// Mitsubishi GX Works2 project: GHEP-Q02U-NEW   PLC: Q02U

// global labels: Global1
VAR_GLOBAL
  Servo_Ready_T AT X40 : BOOL;
  Servo_Ready_X1 AT X41 : BOOL;
  Servo_Ready_X2 AT X42 : BOOL;
  Servo_Ready_Ms AT X43 : BOOL;
  Servo_Ready_S AT X44 : BOOL;
  Physical_Start_PB AT X45 : BOOL;
  Physical_Stop_PB AT X46 : BOOL;
  Physical_Inc_PB AT X47 : BOOL;
  Physical_Dec_PB AT X48 : BOOL;
  Physical_Jog_PB AT X49 : BOOL;
  Sensor_Rev_M AT X4A : BOOL;
  Sensor_Rev_U AT X4B : BOOL;
  Pen1_Toggle_PB AT X4C : BOOL;
  Pen2_Toggle_PB AT X4D : BOOL;
  Switch_Hold_M AT X4E : BOOL;
  Switch_Hold_U AT X4F : BOOL;
  Servo_ON_T AT Y50 : BOOL;
  Servo_ON_X1 AT Y51 : BOOL;
  Servo_ON_X2 AT Y52 : BOOL;
  Servo_ON_Ms AT Y53 : BOOL;
  Servo_ON_S AT Y54 : BOOL;
  DO_Pen1 AT Y55 : BOOL;
  DO_Pen2 AT Y56 : BOOL;
  DO_Alarm_Horn AT Y57 : BOOL;
  Tower_Light_Green AT Y58 : BOOL;
  Tower_Light_Yellow AT Y59 : BOOL;
  Tower_Light_Red AT Y5A : BOOL;
  HMI_Auto_Mode AT M0 : BOOL;
  HMI_Reset_Error AT M1 : BOOL;
  HMI_Start AT M2 : BOOL;
  HMI_Stop AT M3 : BOOL;
  HMI_Reset_Length AT M4 : BOOL;
  HMI_Reset_Roll_T AT M5 : BOOL;
  HMI_Reset_Roll_M AT M6 : BOOL;
  HMI_Reset_Roll_U AT M7 : BOOL;
  HMI_Reset_All_Rolls AT M8 : BOOL;
  HMI_PID_Enable AT M9 : BOOL;
  HMI_Inc_Hold AT M10 : BOOL;
  HMI_Dec_Hold AT M11 : BOOL;
  HMI_Pen1_Cmd AT M12 : BOOL;
  HMI_Pen2_Cmd AT M13 : BOOL;
  HMI_Jog_Crawl_Cmd AT M14 : BOOL;
  HMI_Cmd_Apply_Recipe AT M15 : BOOL;
  HMI_Cmd_Save_Recipe AT M16 : BOOL;
  Zero_Set_T AT M20 : BOOL;
  Zero_Set_X1 AT M21 : BOOL;
  Zero_Set_M AT M22 : BOOL;
  Zero_Set_U AT M23 : BOOL;
  Calib_Set_T AT M24 : BOOL;
  Calib_Set_X1 AT M25 : BOOL;
  Calib_Set_M AT M26 : BOOL;
  Calib_Set_U AT M27 : BOOL;
  HMI_Cmd_Zero_Set AT M28 : BOOL;
  HMI_Cmd_Calib_Set AT M29 : BOOL;
  HMI_Test_T AT M30 : BOOL;
  HMI_Test_X1 AT M31 : BOOL;
  HMI_Test_X2 AT M32 : BOOL;
  HMI_Test_Ms AT M33 : BOOL;
  HMI_Test_S AT M34 : BOOL;
  HMI_Test_M AT M35 : BOOL;
  HMI_Test_U AT M36 : BOOL;
  HMI_Cmd_AutoTune AT M40 : BOOL;
  HMI_Cmd_Save_PID AT M41 : BOOL;
  HMI_Status_AT_Busy AT M42 : BOOL;
  HMI_Status_AT_Done AT M43 : BOOL;
  Servo_Not_Ready_Fault AT M50 : BOOL;
  Hold_Torque_Stop_M AT M51 : BOOL;
  Hold_Torque_Stop_U AT M52 : BOOL;
  Pen1_State AT M53 : BOOL;
  Pen2_State AT M54 : BOOL;
  Pen_Auto_Engaged AT M55 : BOOL;
  Auto_Decel_Flag AT M56 : BOOL;
  State_Machine AT D0 : INT;
  HMI_Status_Text_Code AT D1 : INT;
  HMI_Recipe_Select AT D2 : INT;
  Prev_Recipe_Select AT D3 : INT;
  Current_Line_MPM AT D10 : REAL;
  Total_Length_Meters AT D12 : REAL;
  Set_Target_Length AT D14 : REAL;
  Effective_SP_T AT D16 : REAL;
  RPM_T AT D50 : REAL;
  RPM_X1 AT D52 : REAL;
  RPM_X2 AT D54 : REAL;
  RPM_Ms AT D56 : REAL;
  RPM_S AT D58 : REAL;
  MPM_T AT D60 : REAL;
  MPM_X1 AT D62 : REAL;
  MPM_X2 AT D64 : REAL;
  MPM_Ms AT D66 : REAL;
  MPM_S AT D68 : REAL;
  Target_Line_MPM AT D100 : REAL;
  Max_Speed_MPM AT D102 : REAL;
  Min_Speed_MPM AT D104 : REAL;
  Release_Pen_Speed_MPM AT D106 : REAL;
  Ramp_Accel_Rate AT D108 : REAL;
  Ramp_Decel_Rate AT D110 : REAL;
  Decel_Distance_Meters AT D112 : REAL;
  SP_Tension_T AT D120 : REAL;
  SP_Tension_X1 AT D122 : REAL;
  SP_Tension_M AT D124 : REAL;
  SP_Tension_U AT D126 : REAL;
  Taper_Percent_T AT D128 : REAL;
  Gear_Ratio_T AT D200 : REAL;
  Gear_Ratio_X1 AT D202 : REAL;
  Gear_Ratio_X2 AT D204 : REAL;
  Gear_Ratio_Ms AT D206 : REAL;
  Gear_Ratio_S AT D208 : REAL;
  Gear_Ratio_U AT D210 : REAL;
  Max_RPM_T AT D212 : REAL;
  Max_RPM_X1 AT D214 : REAL;
  Max_RPM_X2 AT D216 : REAL;
  Max_RPM_Ms AT D218 : REAL;
  Max_RPM_S AT D220 : REAL;
  Dia_X1_Roller_mm AT D222 : REAL;
  Dia_X2_Roller_mm AT D224 : REAL;
  Dia_Ms_Roller_mm AT D226 : REAL;
  Dia_S_Roller_mm AT D228 : REAL;
  Core_Dia_T_mm AT D230 : REAL;
  Core_Dia_M_mm AT D232 : REAL;
  Core_Dia_U_mm AT D234 : REAL;
  Max_Dia_T_mm AT D236 : REAL;
  Max_Dia_M_mm AT D238 : REAL;
  Max_Dia_U_mm AT D240 : REAL;
  Speed_Ratio_T AT D250 : REAL;
  Speed_Ratio_X1 AT D252 : REAL;
  Speed_Ratio_Ms AT D254 : REAL;
  Speed_Ratio_S AT D256 : REAL;
  Speed_Offset_X1 AT D260 : REAL;
  Speed_Offset_Ms AT D262 : REAL;
  Speed_Offset_S AT D264 : REAL;
  Min_Torque_M AT D270 : REAL;
  Max_Torque_M AT D272 : REAL;
  Init_Holding_Torque_M AT D274 : REAL;
  Min_Torque_U AT D276 : REAL;
  Max_Torque_U AT D278 : REAL;
  Init_Holding_Torque_U AT D280 : REAL;
  Gear_Ratio_M AT D282 : REAL;
  PPR_Encoder AT D290 : DINT;
  Zero_Offset_T AT D300 : REAL;
  Zero_Offset_X1 AT D302 : REAL;
  Zero_Offset_M AT D304 : REAL;
  Zero_Offset_U AT D306 : REAL;
  Calib_Gain_T AT D310 : REAL;
  Calib_Gain_X1 AT D312 : REAL;
  Calib_Gain_M AT D314 : REAL;
  Calib_Gain_U AT D316 : REAL;
  Weight_Net_T AT D320 : REAL;
  Weight_Net_X1 AT D322 : REAL;
  Weight_Net_M AT D324 : REAL;
  Weight_Net_U AT D326 : REAL;
  Real_Dia_T_mm AT D330 : REAL;
  Real_Dia_M_mm AT D332 : REAL;
  Real_Dia_U_mm AT D334 : REAL;
  Kp_T AT D340 : REAL;
  Ki_T AT D342 : REAL;
  Kd_T AT D344 : REAL;
  Kp_X1 AT D346 : REAL;
  Ki_X1 AT D348 : REAL;
  Kd_X1 AT D350 : REAL;
  Kp_X2 AT D352 : REAL;
  Ki_X2 AT D354 : REAL;
  Kd_X2 AT D356 : REAL;
  Kp_Ms AT D358 : REAL;
  Ki_Ms AT D360 : REAL;
  Kd_Ms AT D362 : REAL;
  Kp_S AT D364 : REAL;
  Ki_S AT D366 : REAL;
  Kd_S AT D368 : REAL;
  Kp_M AT D370 : REAL;
  Ki_M AT D372 : REAL;
  Kd_M AT D374 : REAL;
  Kp_U AT D376 : REAL;
  Ki_U AT D378 : REAL;
  Kd_U AT D380 : REAL;
  Curr_Pulse_T AT D520 : DINT;
  Curr_Pulse_X1 AT D522 : DINT;
  Curr_Pulse_X2 AT D524 : DINT;
  Curr_Pulse_Ms AT D526 : DINT;
  HMI_Axis_Select AT D600 : INT;
  HMI_Disp_Kp AT D602 : REAL;
  HMI_Disp_Ki AT D604 : REAL;
  HMI_Disp_Kd AT D606 : REAL;
  HMI_Disp_Calib_Gain AT D608 : REAL;
  HMI_Disp_Zero_Offset AT D610 : REAL;
  Test_Speed_T AT D620 : REAL;
  Test_Torque_T AT D622 : REAL;
  Test_Speed_X1 AT D624 : REAL;
  Test_Speed_X2 AT D626 : REAL;
  Test_Speed_Ms AT D628 : REAL;
  Test_Speed_S AT D630 : REAL;
  Test_Torque_M AT D632 : REAL;
  Test_Speed_U AT D634 : REAL;
END_VAR

// task Task_01 (event TRUE, interval 0, priority 31): POU_01
// task POU_INIT (event TRUE, interval 0, priority 31): POU_INIT

PROGRAM POU_01
VAR
  Delta_T : DINT;  (* Chenh lech xung Truc Thu T *)
  Delta_X1 : DINT;  (* Chenh lech xung Truc Keo X1 *)
  Delta_X2 : DINT;  (* Chenh lech xung Master X2 *)
  Delta_Ms : DINT;  (* Chenh lech xung Truc Ghep Ms *)
  Delta_Pulse_X2 : DINT;  (* Chenh lech xung Master X2 tinh chieu dai mang *)
  Prev_Pulse_T : DINT;  (* Xung Truc T chu ky truoc *)
  Prev_Pulse_X1 : DINT;  (* Xung Truc X1 chu ky truoc *)
  Prev_Pulse_X2 : DINT;  (* Xung Truc X2 chu ky truoc *)
  Prev_Pulse_Ms : DINT;  (* Xung Truc Ms chu ky truoc *)
  Total_PPR : DINT;  (* Tong xung sau khi nhan 4 *)
  Raw_Analog_S : REAL;  (* Gia tri tho Analog Speed Servo S *)
  Raw_RPM_T : REAL;  (* Toc do RPM tho Truc Thu T *)
  Raw_RPM_X1 : REAL;  (* Toc do RPM tho Truc Keo X1 *)
  Raw_RPM_X2 : REAL;  (* Toc do RPM tho Truc Master X2 *)
  Raw_RPM_Ms : REAL;  (* Toc do RPM tho Truc Ghep Ms *)
  Raw_RPM_S : REAL;  (* Toc do RPM tho Truc Dau S *)
  Buf_RPM_T_1 : REAL;  (* Buffer mau 1 loc trung binh trượt T *)
  Buf_RPM_T_2 : REAL;  (* Buffer mau 2 loc trung binh trượt T *)
  Buf_RPM_T_3 : REAL;  (* Buffer mau 3 loc trung binh trượt T *)
  Buf_RPM_X1_1 : REAL;  (* Buffer mau 1 loc trung binh trượt X1 *)
  Buf_RPM_X1_2 : REAL;  (* Buffer mau 2 loc trung binh trượt X1 *)
  Buf_RPM_X1_3 : REAL;  (* Buffer mau 3 loc trung binh trượt X1 *)
  Buf_RPM_X2_1 : REAL;  (* Buffer mau 1 loc trung binh trượt X2 *)
  Buf_RPM_X2_2 : REAL;  (* Buffer mau 2 loc trung binh trượt X2 *)
  Buf_RPM_X2_3 : REAL;  (* Buffer mau 3 loc trung binh trượt X2 *)
  Buf_RPM_Ms_1 : REAL;  (* Buffer mau 1 loc trung binh trượt Ms *)
  Buf_RPM_Ms_2 : REAL;  (* Buffer mau 2 loc trung binh trượt Ms *)
  Buf_RPM_Ms_3 : REAL;  (* Buffer mau 3 loc trung binh trượt Ms *)
  Buf_RPM_S_1 : REAL;  (* Buffer mau 1 loc trung binh trượt S *)
  Buf_RPM_S_2 : REAL;  (* Buffer mau 2 loc trung binh trượt S *)
  Buf_RPM_S_3 : REAL;  (* Buffer mau 3 loc trung binh trượt S *)
  ADC_CH1_Raw : INT;  (* Gia tri tho ADC CH1 Loadcell T *)
  ADC_CH2_Raw : INT;  (* Gia tri tho ADC CH2 Loadcell X1 *)
  ADC_CH3_Raw : INT;  (* Gia tri tho ADC CH3 Loadcell M *)
  ADC_CH4_Raw : INT;  (* Gia tri tho ADC CH4 Loadcell U *)
  ADC_CH5_Raw : INT;  (* Gia tri tho ADC CH5 Analog Servo S *)
  ADC_CH6_Raw : INT;  (* Gia tri tho ADC CH6 Du phong *)
  ADC_CH7_Raw : INT;  (* Gia tri tho ADC CH7 Du phong *)
  ADC_CH8_Raw : INT;  (* Gia tri tho ADC CH8 Du phong *)
  Cmd_Start : BOOL;  (* Lenh tong hop Start chay may *)
  Cmd_Stop : BOOL;  (* Lenh tong hop Stop dung may *)
  Cmd_Inc : BOOL;  (* Lenh tong hop Tang toc *)
  Cmd_Dec : BOOL;  (* Lenh tong hop Giam toc *)
  Cmd_Jog_Crawl : BOOL;  (* Lenh tong hop Bo cham luon mang *)
  Trig_Pen1 : BOOL;  (* Xung kich toggle Pen 1 *)
  Prev_Pen1_PB : BOOL;  (* Trang thai Pen 1 chu ky truoc *)
  Trig_Pen2 : BOOL;  (* Xung kich toggle Pen 2 *)
  Prev_Pen2_PB : BOOL;  (* Trang thai Pen 2 chu ky truoc *)
  Pen1_Next_State : BOOL;  (* Trang thai tiep theo Pen 1 *)
  Pen2_Next_State : BOOL;  (* Trang thai tiep theo Pen 2 *)
  Trig_X50 : BOOL;  (* Xung kich sensor cuon M *)
  Prev_X50 : BOOL;  (* Trang thai sensor cuon M chu ky truoc *)
  Trig_X51 : BOOL;  (* Xung kich sensor cuon U *)
  Prev_X51 : BOOL;  (* Trang thai sensor cuon U chu ky truoc *)
  Trig_PID_10ms : BOOL;  (* Xung kich nhap PID 10ms *)
  Prev_SM409 : BOOL;  (* Trang thai SM409 chu ky truoc *)
  Inc_Hold_Timer : INT;  (* Timer giu nut tang toc *)
  Dec_Hold_Timer : INT;  (* Timer giu nut giam toc *)
  Dynamic_Accel_Step : REAL;  (* Buoc tang giam toc luy tien *)
  Last_Pulse_X2_Len : DINT;  (* Xung X2 chu ky truoc tinh chieu dai *)
  Last_Pulse_X2_T : DINT;  (* Xung X2 chu ky truoc tinh duong kinh T *)
  Last_Pulse_X2_M : DINT;  (* Xung X2 chu ky truoc tinh duong kinh M *)
  Last_Pulse_X2_U : DINT;  (* Xung X2 chu ky truoc tinh duong kinh U *)
  Last_Pulse_T : DINT;  (* Xung T chu ky truoc *)
  Rev_Count_T : DINT;  (* So vong quay cuon Thu T *)
  Rev_Count_M : DINT;  (* So vong quay cuon Thang M *)
  Rev_Count_U : DINT;  (* So vong quay cuon Xa U *)
  Accum_Length_mm : REAL;  (* Chieu dai tich luy mm *)
  Delta_Length_mm : REAL;  (* Chieu dai di duoc trong 1 scan mm *)
  Raw_Dia_T_mm : REAL;  (* Duong kinh tho tinh toan T mm *)
  Raw_Dia_M_mm : REAL;  (* Duong kinh tho tinh toan M mm *)
  Raw_Dia_U_mm : REAL;  (* Duong kinh tho tinh toan U mm *)
  Base_Speed_X2 : REAL;  (* Toc do co ban theo Master X2 (0..16000) *)
  SP_Speed_X2 : REAL;  (* Setpoint toc do Master X2 *)
  SP_Speed_X1 : REAL;  (* Setpoint toc do Keo X1 *)
  SP_Speed_Ms : REAL;  (* Setpoint toc do Ghep Ms *)
  SP_Speed_S : REAL;  (* Setpoint toc do Dau S *)
  SP_Speed_T : REAL;  (* Setpoint toc do Thu T *)
  Feedback_Speed_X2 : REAL;  (* Feedback toc do Master X2 *)
  Feedback_Speed_Ms : REAL;  (* Feedback toc do Ghep Ms *)
  Feedback_Speed_S : REAL;  (* Feedback toc do Dau S (tu Analog Out Servo) *)
  PID_Out_X2 : REAL;  (* Ngo ra PID Master X2 *)
  PID_Out_Ms : REAL;  (* Ngo ra PID Ghep Ms *)
  PID_Out_S : REAL;  (* Ngo ra PID Dau S *)
  PID_Out_X1 : REAL;  (* Ngo ra PID Keo X1 *)
  PID_Out_T : REAL;  (* Ngo ra PID Thu T *)
  PID_Out_M : REAL;  (* Ngo ra PID Thang M *)
  PID_Out_U : REAL;  (* Ngo ra PID Xa U *)
  Calc_Speed_X2 : REAL;  (* Toc do tong hop xuat DAC Master X2 *)
  Calc_Speed_X1 : REAL;  (* Toc do tong hop xuat DAC Keo X1 *)
  Calc_Speed_Ms : REAL;  (* Toc do tong hop xuat DAC Ghep Ms *)
  Calc_Speed_S : REAL;  (* Toc do tong hop xuat DAC Dau S *)
  Calc_Speed_T : REAL;  (* Toc do tong hop xuat DAC Thu T *)
  Calc_Speed_U : REAL;  (* Toc do tong hop xuat DAC Xa U *)
  Calc_Torque_T : REAL;  (* Torque tong hop xuat DAC Thu T *)
  Calc_Torque_M : REAL;  (* Torque tong hop xuat DAC Thang M *)
  Base_Torque_M : REAL;  (* Torque co ban 3 pha Thang M (%) *)
  pid_X2 : FB_TENSION_PID;  (* Instance PID Master X2 *)
  pid_Ms : FB_TENSION_PID;  (* Instance PID Ghep Ms *)
  pid_S : FB_TENSION_PID;  (* Instance PID Dau S *)
  pid_X1 : FB_TENSION_PID;  (* Instance PID Keo X1 *)
  pid_T : FB_TENSION_PID;  (* Instance PID Thu T *)
  pid_M : FB_TENSION_PID;  (* Instance PID Thang M *)
  pid_U : FB_TENSION_PID;  (* Instance PID Xa U *)
END_VAR
(* ============================================================================ *)
(* MÃ NGUỒN POU_01: HỆ THỐNG MÁY GHÉP MÀNG METALIZE TỰ ĐỘNG - MITSUBISHI Q02U  *)
(* BẢO VỆ TOÀN DIỆN CHỐNG LỖI 4140 OPERATION ERROR (CHIA CHO 0 & TRÀN SỐ DINT)  *)
(* CẤU HÌNH PHẦN CỨNG:                                                          *)
(*   - Slot 0 (H00): Q68ADV (8CH Analog In: Loadcell T, X1, M, U & Analog S)    *)
(*   - Slot 1 (H10): Q68DAV (8CH Analog Out: Speed/Torque T, X1, X2, Ms, S, M, U) *)
(*   - Slot 2 (H20): QD62D  (2CH High Speed Counter: CH1=Trục T, CH2=Trục X1)  *)
(*   - Slot 3 (H30): QD62D  (2CH High Speed Counter: CH1=Trục X2, CH2=Trục Ms) *)
(*   - Slot 4 (H40): QX40   (16CH Digital Input: X40..X4F)                     *)
(*   - Slot 5 (H50): QY40   (16CH Digital Output: Y50..Y5F)                    *)
(*   - Slot 6 (H60): QJ71C24N (RS232/RS485 Serial)                             *)
(* ============================================================================ *)

(* ============================================================================ *)
(* 0. KIỂM TRA & GÁN GIÁ TRỊ AN TOÀN TRÁNH CHIA CHO 0 (ZERO DIV PROTECTION)    *)
(* ============================================================================ *)
IF PPR_Encoder      <= 0     THEN PPR_Encoder      := 2000;  END_IF;
IF Max_RPM_X2       <= 0.0   THEN Max_RPM_X2       := 1000.0; END_IF;
IF Max_RPM_X1       <= 0.0   THEN Max_RPM_X1       := 1000.0; END_IF;
IF Max_RPM_Ms       <= 0.0   THEN Max_RPM_Ms       := 3000.0; END_IF;
IF Max_RPM_S        <= 0.0   THEN Max_RPM_S        := 3000.0; END_IF;
IF Max_RPM_T        <= 0.0   THEN Max_RPM_T        := 1500.0; END_IF;

IF Gear_Ratio_T     <= 0.0   THEN Gear_Ratio_T     := 10.1;  END_IF;
IF Gear_Ratio_X1    <= 0.0   THEN Gear_Ratio_X1    := 8.0;   END_IF;
IF Gear_Ratio_X2    <= 0.0   THEN Gear_Ratio_X2    := 8.0;   END_IF;
IF Gear_Ratio_Ms    <= 0.0   THEN Gear_Ratio_Ms    := 10.0;  END_IF;
IF Gear_Ratio_S     <= 0.0   THEN Gear_Ratio_S     := 10.0;  END_IF;
IF Gear_Ratio_U     <= 0.0   THEN Gear_Ratio_U     := 1.0;     END_IF; (* Xả U: 1.0 : 1 *)
IF Gear_Ratio_M     <= 0.0   THEN Gear_Ratio_M     := 1.03125; END_IF; (* Trục Xả Metalize M: Gear = 33/32 = 1.03125 *)

IF Dia_X1_Roller_mm <= 0.0   THEN Dia_X1_Roller_mm := 300.5; END_IF;
IF Dia_X2_Roller_mm <= 0.0   THEN Dia_X2_Roller_mm := 300.5; END_IF;
IF Dia_Ms_Roller_mm <= 0.0   THEN Dia_Ms_Roller_mm := 200.0; END_IF;
IF Dia_S_Roller_mm  <= 0.0   THEN Dia_S_Roller_mm  := 100.0; END_IF;

IF Core_Dia_T_mm    <= 0.0   THEN Core_Dia_T_mm    := 76.0;   END_IF;
IF Core_Dia_M_mm    <= 0.0   THEN Core_Dia_M_mm    := 76.0;   END_IF;
IF Core_Dia_U_mm    <= 0.0   THEN Core_Dia_U_mm    := 76.0;   END_IF;

IF Max_Dia_T_mm     <= 0.0   THEN Max_Dia_T_mm     := 1000.0; END_IF;
IF Max_Dia_M_mm     <= 0.0   THEN Max_Dia_M_mm     := 600.0;  END_IF;
IF Max_Dia_U_mm     <= 0.0   THEN Max_Dia_U_mm     := 800.0;  END_IF;

IF Real_Dia_T_mm    < Core_Dia_T_mm THEN Real_Dia_T_mm := Core_Dia_T_mm; END_IF;
IF Real_Dia_M_mm    < Core_Dia_M_mm THEN Real_Dia_M_mm := Max_Dia_M_mm;  END_IF;
IF Real_Dia_U_mm    < Core_Dia_U_mm THEN Real_Dia_U_mm := Max_Dia_U_mm;  END_IF;

IF Max_Speed_MPM    <= 0.0   THEN Max_Speed_MPM    := 100.0;  END_IF;
IF Min_Speed_MPM    <= 0.0   THEN Min_Speed_MPM    := 2.0;    END_IF;
IF Ramp_Accel_Rate  <= 0.0   THEN Ramp_Accel_Rate  := 0.5;    END_IF;
IF Ramp_Decel_Rate  <= 0.0   THEN Ramp_Decel_Rate  := 1.0;    END_IF;

(* ============================================================================ *)
(* 1. KÍCH HOẠT VÀ ĐỌC 4 KÊNH ENCODER QD62D (SLOT 2 & 3) MỖI SCAN               *)
(* ============================================================================ *)
(* Kích hoạt cờ đếm xung cho 2 module QD62D *)
Y21 := TRUE; (* QD62D #1 (Slot 2 H20) CH1: Enable Trục Thu T *)
Y22 := TRUE; (* QD62D #1 (Slot 2 H20) CH2: Enable Trục Kéo X1 *)
Y31 := TRUE; (* QD62D #2 (Slot 3 H30) CH1: Enable Trục Master X2 *)
Y32 := TRUE; (* QD62D #2 (Slot 3 H30) CH2: Enable Trục Ghép Ms *)

(* Đọc xung 32-bit từ Buffer Memory QD62D liên tục mỗi scan *)
DMOV(TRUE, U2\G2,  Curr_Pulse_T);  (* Slot 2 CH1: Trục Thu T *)
DMOV(TRUE, U2\G10, Curr_Pulse_X1); (* Slot 2 CH2: Trục Kéo X1 *)
DMOV(TRUE, U3\G2,  Curr_Pulse_X2); (* Slot 3 CH1: Trục Master X2 *)
DMOV(TRUE, U3\G10, Curr_Pulse_Ms); (* Slot 3 CH2: Trục Ghép Ms *)

(* ============================================================================ *)
(* 2. ĐỌC VÀ LỌC 8 KÊNH ANALOG INPUT TỪ MODULE Q68ADV (SLOT 0 - U0\G1..U0\G8)   *)
(* ============================================================================ *)
ADC_CH1_Raw := U0\G1; (* Loadcell Lực căng Thu T *)
ADC_CH2_Raw := U0\G2; (* Loadcell Lực căng Kéo X1 *)
ADC_CH3_Raw := U0\G3; (* Loadcell Lực căng Thắng M *)
ADC_CH4_Raw := U0\G4; (* Loadcell Lực căng Xả U *)
ADC_CH5_Raw := U0\G5; (* Tín hiệu Analog Out Tốc độ Servo Trục S *)
ADC_CH6_Raw := U0\G6; (* Dự phòng CH6 *)
ADC_CH7_Raw := U0\G7; (* Dự phòng CH7 *)
ADC_CH8_Raw := U0\G8; (* Dự phòng CH8 *)

(* Chuyển sang thanh ghi hiển thị D500..D507 *)
D500 := INT_TO_WORD(ADC_CH1_Raw);
D501 := INT_TO_WORD(ADC_CH2_Raw);
D502 := INT_TO_WORD(ADC_CH3_Raw);
D503 := INT_TO_WORD(ADC_CH4_Raw);
D504 := INT_TO_WORD(ADC_CH5_Raw);
D505 := INT_TO_WORD(ADC_CH6_Raw);
D506 := INT_TO_WORD(ADC_CH7_Raw);
D507 := INT_TO_WORD(ADC_CH8_Raw);

(* Tính giá trị Lực căng thực tế (kg) sau khi trừ Zero Offset và nhân Gain Calib *)
IF Calib_Gain_T <= 0.0 THEN Calib_Gain_T := 1.0; END_IF;
Weight_Net_T := ((INT_TO_REAL(ADC_CH1_Raw) - Zero_Offset_T) * Calib_Gain_T * 50.0) / 16000.0;
IF Weight_Net_T < 0.0 THEN Weight_Net_T := 0.0; END_IF;

IF Calib_Gain_X1 <= 0.0 THEN Calib_Gain_X1 := 1.0; END_IF;
Weight_Net_X1 := ((INT_TO_REAL(ADC_CH2_Raw) - Zero_Offset_X1) * Calib_Gain_X1 * 50.0) / 16000.0;
IF Weight_Net_X1 < 0.0 THEN Weight_Net_X1 := 0.0; END_IF;

IF Calib_Gain_M <= 0.0 THEN Calib_Gain_M := 1.0; END_IF;
Weight_Net_M := ((INT_TO_REAL(ADC_CH3_Raw) - Zero_Offset_M) * Calib_Gain_M * 50.0) / 16000.0;
IF Weight_Net_M < 0.0 THEN Weight_Net_M := 0.0; END_IF;

IF Calib_Gain_U <= 0.0 THEN Calib_Gain_U := 1.0; END_IF;
Weight_Net_U := ((INT_TO_REAL(ADC_CH4_Raw) - Zero_Offset_U) * Calib_Gain_U * 50.0) / 16000.0;
IF Weight_Net_U < 0.0 THEN Weight_Net_U := 0.0; END_IF;

(* Xử lý Nút Set Zero Lực căng *)
IF Zero_Set_T OR (HMI_Cmd_Zero_Set AND HMI_Axis_Select = 1) THEN
    Zero_Offset_T := INT_TO_REAL(ADC_CH1_Raw);
    Zero_Set_T    := FALSE;
END_IF;
IF Zero_Set_X1 OR (HMI_Cmd_Zero_Set AND HMI_Axis_Select = 2) THEN
    Zero_Offset_X1 := INT_TO_REAL(ADC_CH2_Raw);
    Zero_Set_X1    := FALSE;
END_IF;
IF Zero_Set_M OR (HMI_Cmd_Zero_Set AND HMI_Axis_Select = 6) THEN
    Zero_Offset_M := INT_TO_REAL(ADC_CH3_Raw);
    Zero_Set_M    := FALSE;
END_IF;
IF Zero_Set_U OR (HMI_Cmd_Zero_Set AND HMI_Axis_Select = 7) THEN
    Zero_Offset_U := INT_TO_REAL(ADC_CH4_Raw);
    Zero_Set_U    := FALSE;
END_IF;
IF HMI_Cmd_Zero_Set THEN
    HMI_Cmd_Zero_Set := FALSE;
END_IF;

(* ============================================================================ *)
(* 3. BẢO VỆ 5 TRỤC SERVO READY TRÊN MODULE QX40 (SLOT 4 - X40..X44)            *)
(* ============================================================================ *)
Servo_Ready_T  := X40; (* Sẵn sàng Servo Thu T *)
Servo_Ready_X1 := X41; (* Sẵn sàng Servo Kéo X1 *)
Servo_Ready_X2 := X42; (* Sẵn sàng Servo Master X2 *)
Servo_Ready_Ms := X43; (* Sẵn sàng Servo Ghép Ms *)
Servo_Ready_S  := X44; (* Sẵn sàng Servo Dầu S *)

Servo_Not_Ready_Fault := NOT(Servo_Ready_T) OR NOT(Servo_Ready_X1) OR NOT(Servo_Ready_X2) OR NOT(Servo_Ready_Ms) OR NOT(Servo_Ready_S);

IF Servo_Not_Ready_Fault AND State_Machine = 1 THEN
    State_Machine := 0; (* Dừng khẩn cấp nếu đang chạy tự động *)
END_IF;

(* ============================================================================ *)
(* 4. ĐỌC NÚT NHẤN, CẢM BIẾN VÀ CÔNG TẮC GẠT TRÊN MODULE QX40 (SLOT 4 - X45..X4F) *)
(* ============================================================================ *)
Physical_Start_PB := X45; (* Nút Start vật lý *)
Physical_Stop_PB  := X46; (* Nút Stop vật lý *)
Physical_Inc_PB   := X47; (* Nút Tăng tốc vật lý *)
Physical_Dec_PB   := X48; (* Nút Giảm tốc vật lý *)
Physical_Jog_PB   := X49; (* Nút Bò chậm luồn màng vật lý *)
Sensor_Rev_M      := X4A; (* Cảm biến tiệm cận đếm vòng cuộn M *)
Sensor_Rev_U      := X4B; (* Cảm biến tiệm cận đếm vòng cuộn U *)
Pen1_Toggle_PB    := X4C; (* Nút nhấn Pen 1 ngoài tủ *)
Pen2_Toggle_PB    := X4D; (* Nút nhấn Pen 2 ngoài tủ *)
Switch_Hold_M     := X4E; (* Công tắc gạt giữ Torque M khi dừng *)
Switch_Hold_U     := X4F; (* Công tắc gạt giữ Torque U khi dừng *)

Hold_Torque_Stop_M := Switch_Hold_M;
Hold_Torque_Stop_U := Switch_Hold_U;

(* ============================================================================ *)
(* 5. QUẢN LÝ CÔNG THỨC ĐƠN HÀNG (RECIPE MANAGEMENT CHO CÔNG NHÂN)             *)
(* ============================================================================ *)
IF HMI_Recipe_Select <= 0 OR HMI_Recipe_Select > 5 THEN
    HMI_Recipe_Select := 2; (* Mặc định chọn Recipe 2: Hàng Tiêu Chuẩn *)
END_IF;

IF (HMI_Recipe_Select <> Prev_Recipe_Select) OR HMI_Cmd_Apply_Recipe THEN
    CASE HMI_Recipe_Select OF
        1: (* 1. HÀNG MÀNG MỎNG (BOPP 12~15 mic - Bao bì bánh kẹo) *)
            Target_Line_MPM  := 45.0;  (* Tốc độ chuẩn 45 m/p *)
            SP_Tension_T     := 12.0;  (* Lực căng Thu T: 12 kg *)
            SP_Tension_X1    := 10.0;  (* Lực căng Kéo X1: 10 kg *)
            SP_Tension_M     := 4.0;   (* Lực căng Thắng Metalize M: 4 kg *)
            SP_Tension_U     := 8.0;   (* Lực căng Xả U: 8 kg *)
            Taper_Percent_T  := 15.0;  (* Giảm côn lực 15% *)
            Ramp_Accel_Rate  := 0.05;  (* Gia tốc êm ái *)
            Ramp_Decel_Rate  := 0.08;

        2: (* 2. HÀNG TIÊU CHUẨN (BOPP 18~20 mic + Giấy 100~150g - Hộp thông dụng) *)
            Target_Line_MPM  := 60.0;  (* Tốc độ chuẩn 60 m/p *)
            SP_Tension_T     := 16.0;  (* Lực căng Thu T: 16 kg *)
            SP_Tension_X1    := 14.0;  (* Lực căng Kéo X1: 14 kg *)
            SP_Tension_M     := 6.0;   (* Lực căng Thắng Metalize M: 6 kg *)
            SP_Tension_U     := 12.0;  (* Lực căng Xả U: 12 kg *)
            Taper_Percent_T  := 20.0;  (* Giảm côn lực 20% *)
            Ramp_Accel_Rate  := 0.08;  (* Gia tốc tiêu chuẩn *)
            Ramp_Decel_Rate  := 0.10;

        3: (* 3. HÀNG GIẤY DÀY / BÌA CỨNG (Duplex / Ivory 250~350g + Metalize) *)
            Target_Line_MPM  := 50.0;  (* Tốc độ chuẩn 50 m/p *)
            SP_Tension_T     := 25.0;  (* Lực căng Thu T: 25 kg *)
            SP_Tension_X1    := 22.0;  (* Lực căng Kéo X1: 22 kg *)
            SP_Tension_M     := 8.0;   (* Lực căng Thắng Metalize M: 8 kg *)
            SP_Tension_U     := 18.0;  (* Lực căng Xả U: 18 kg *)
            Taper_Percent_T  := 25.0;  (* Giảm côn lực 25% *)
            Ramp_Accel_Rate  := 0.06;
            Ramp_Decel_Rate  := 0.10;

        4: (* 4. HÀNG MÀNG NHÔM / FOIL DẺO CAO CẤP (Alu Foil 9~12 mic / PET) *)
            Target_Line_MPM  := 40.0;  (* Tốc độ chuẩn 40 m/p *)
            SP_Tension_T     := 10.0;  (* Lực căng Thu T: 10 kg *)
            SP_Tension_X1    := 8.0;   (* Lực căng Kéo X1: 8 kg *)
            SP_Tension_M     := 3.5;   (* Lực căng Thắng Metalize M: 3.5 kg *)
            SP_Tension_U     := 7.0;   (* Lực căng Xả U: 7 kg *)
            Taper_Percent_T  := 15.0;
            Ramp_Accel_Rate  := 0.04;  (* Gia tốc siêu êm chống đứt foil *)
            Ramp_Decel_Rate  := 0.06;

        5: (* 5. CHẾ ĐỘ TÙY CHỈNH (CUSTOM) *)
            Target_Line_MPM := Target_Line_MPM;
    END_CASE;
    Prev_Recipe_Select   := HMI_Recipe_Select;
    HMI_Cmd_Apply_Recipe := FALSE;
END_IF;

IF HMI_Cmd_Save_Recipe THEN
    HMI_Recipe_Select    := 5;
    Prev_Recipe_Select   := 5;
    HMI_Cmd_Save_Recipe  := FALSE;
END_IF;

(* ============================================================================ *)
(* 6. NẠP LẠI ĐƯỜNG KÍNH CUỘN TỪ HMI & NÚT THAY CUỘN MỚI TOÀN BỘ 1-CLICK        *)
(* ============================================================================ *)
IF HMI_Reset_All_Rolls THEN
    Real_Dia_T_mm       := Core_Dia_T_mm; (* Thu T về lõi *)
    Real_Dia_M_mm       := Max_Dia_M_mm;  (* Thắng M về cuộn đầy *)
    Real_Dia_U_mm       := Max_Dia_U_mm;  (* Xả U về cuộn đầy *)
    Total_Length_Meters := 0.0;           (* Xóa mét về 0 *)
    Accum_Length_mm     := 0.0;
    HMI_Reset_All_Rolls := FALSE;
END_IF;
IF HMI_Reset_Roll_T THEN Real_Dia_T_mm := Core_Dia_T_mm; HMI_Reset_Roll_T := FALSE; END_IF;
IF HMI_Reset_Roll_M THEN Real_Dia_M_mm := Max_Dia_M_mm;  HMI_Reset_Roll_M := FALSE; END_IF;
IF HMI_Reset_Roll_U THEN Real_Dia_U_mm := Max_Dia_U_mm;  HMI_Reset_Roll_U := FALSE; END_IF;

(* ============================================================================ *)
(* 7. TỔNG HỢP NÚT NHẤN HMI & NÚT NHẤN VẬT LÝ                                  *)
(* ============================================================================ *)
Cmd_Start     := HMI_Start OR Physical_Start_PB;
Cmd_Stop      := HMI_Stop OR Physical_Stop_PB OR Servo_Not_Ready_Fault;
Cmd_Inc       := HMI_Inc_Hold OR Physical_Inc_PB;
Cmd_Dec       := HMI_Dec_Hold OR Physical_Dec_PB;
Cmd_Jog_Crawl := HMI_Jog_Crawl_Cmd OR Physical_Jog_PB;

(* ============================================================================ *)
(* 8. ĐIỀU KHIỂN 2 PEN ÉP MÀNG (SINGLE-COIL LOGIC)                             *)
(* ============================================================================ *)
Trig_Pen1 := (Pen1_Toggle_PB AND NOT(Prev_Pen1_PB)) OR HMI_Pen1_Cmd;
Prev_Pen1_PB := Pen1_Toggle_PB;
IF HMI_Pen1_Cmd THEN HMI_Pen1_Cmd := FALSE; END_IF;

Trig_Pen2 := (Pen2_Toggle_PB AND NOT(Prev_Pen2_PB)) OR HMI_Pen2_Cmd;
Prev_Pen2_PB := Pen2_Toggle_PB;
IF HMI_Pen2_Cmd THEN HMI_Pen2_Cmd := FALSE; END_IF;

IF State_Machine = 1 AND Current_Line_MPM >= 5.0 AND NOT Pen_Auto_Engaged THEN
    Pen1_Next_State := TRUE;
    Pen2_Next_State := TRUE;
ELSIF (State_Machine = 0 OR Current_Line_MPM <= Release_Pen_Speed_MPM) AND NOT (Trig_Pen1 OR Trig_Pen2) THEN
    Pen1_Next_State := FALSE;
    Pen2_Next_State := FALSE;
ELSE
    IF Trig_Pen1 THEN Pen1_Next_State := NOT Pen1_State; ELSE Pen1_Next_State := Pen1_State; END_IF;
    IF Trig_Pen2 THEN Pen2_Next_State := NOT Pen2_State; ELSE Pen2_Next_State := Pen2_State; END_IF;
END_IF;

Pen1_State := Pen1_Next_State;
Pen2_State := Pen2_Next_State;
Pen_Auto_Engaged := (State_Machine = 1 AND Current_Line_MPM >= 5.0);

(* ============================================================================ *)
(* 9. TĂNG GIẢM TỐC LŨY TIẾN THEO THỜI GIAN GIỮ PHÍM INC / DEC                 *)
(* ============================================================================ *)
IF Cmd_Inc THEN
    Inc_Hold_Timer := Inc_Hold_Timer + 1;
    IF Inc_Hold_Timer < 50 THEN
        Dynamic_Accel_Step := Ramp_Accel_Rate;
    ELSIF Inc_Hold_Timer < 150 THEN
        Dynamic_Accel_Step := Ramp_Accel_Rate * 2.0;
    ELSE
        Dynamic_Accel_Step := Ramp_Accel_Rate * 5.0;
    END_IF;
    Target_Line_MPM := Target_Line_MPM + Dynamic_Accel_Step;
    IF Target_Line_MPM > Max_Speed_MPM THEN Target_Line_MPM := Max_Speed_MPM; END_IF;
ELSE
    Inc_Hold_Timer := 0;
END_IF;

IF Cmd_Dec THEN
    Dec_Hold_Timer := Dec_Hold_Timer + 1;
    IF Dec_Hold_Timer < 50 THEN
        Dynamic_Accel_Step := Ramp_Decel_Rate;
    ELSIF Dec_Hold_Timer < 150 THEN
        Dynamic_Accel_Step := Ramp_Decel_Rate * 2.0;
    ELSE
        Dynamic_Accel_Step := Ramp_Decel_Rate * 5.0;
    END_IF;
    Target_Line_MPM := Target_Line_MPM - Dynamic_Accel_Step;
    IF Target_Line_MPM < Min_Speed_MPM THEN Target_Line_MPM := Min_Speed_MPM; END_IF;
ELSE
    Dec_Hold_Timer := 0;
END_IF;

(* Ramping tốc độ hiện tại *)
IF Current_Line_MPM < Target_Line_MPM THEN
    Current_Line_MPM := Current_Line_MPM + Ramp_Accel_Rate;
    IF Current_Line_MPM > Target_Line_MPM THEN Current_Line_MPM := Target_Line_MPM; END_IF;
ELSIF Current_Line_MPM > Target_Line_MPM THEN
    Current_Line_MPM := Current_Line_MPM - Ramp_Decel_Rate;
    IF Current_Line_MPM < Target_Line_MPM THEN Current_Line_MPM := Target_Line_MPM; END_IF;
END_IF;

(* ============================================================================ *)
(* 10. TÍNH ĐƯỜNG KÍNH 3 CUỘN T, M, U VÀ ĐO CHIỀU DÀI MÀNG CHẠY TỪ ENCODER X2   *)
(* ============================================================================ *)
Delta_Pulse_X2 := ABS(Curr_Pulse_X2 - Last_Pulse_X2_Len);

IF Delta_Pulse_X2 > 0 AND State_Machine = 1 AND Total_PPR > 0 THEN
    Delta_Length_mm := (DINT_TO_REAL(Delta_Pulse_X2) * 3.1415 * Dia_X2_Roller_mm) / (DINT_TO_REAL(Total_PPR) * Gear_Ratio_X2);
    Accum_Length_mm := Accum_Length_mm + Delta_Length_mm;
    
    IF Accum_Length_mm >= 1000.0 THEN
        Total_Length_Meters := Total_Length_Meters + (Accum_Length_mm / 1000.0);
        Accum_Length_mm     := 0.0;
    END_IF;
END_IF;
Last_Pulse_X2_Len := Curr_Pulse_X2;

IF HMI_Reset_Length THEN
    Total_Length_Meters := 0.0;
    Accum_Length_mm     := 0.0;
    HMI_Reset_Length    := FALSE;
END_IF;

(* Đường kính cuộn Thu T theo xung Master X2 *)
IF Total_PPR > 0 AND (Curr_Pulse_T - Last_Pulse_T) >= REAL_TO_DINT(DINT_TO_REAL(Total_PPR) * Gear_Ratio_T) THEN
    Rev_Count_T := Rev_Count_T + 1;
    IF (Curr_Pulse_X2 - Last_Pulse_X2_T) > 0 THEN
        Raw_Dia_T_mm := (DINT_TO_REAL(Curr_Pulse_X2 - Last_Pulse_X2_T) * Dia_X2_Roller_mm) / (DINT_TO_REAL(Total_PPR) * Gear_Ratio_X2);
        IF Raw_Dia_T_mm < Core_Dia_T_mm THEN Raw_Dia_T_mm := Core_Dia_T_mm; END_IF;
        IF Raw_Dia_T_mm > Max_Dia_T_mm THEN Raw_Dia_T_mm := Max_Dia_T_mm; END_IF;
        Real_Dia_T_mm := Real_Dia_T_mm + ((Raw_Dia_T_mm - Real_Dia_T_mm) * 0.2);
    END_IF;
    Last_Pulse_X2_T := Curr_Pulse_X2;
    Last_Pulse_T    := Curr_Pulse_T;
END_IF;

(* Đường kính cuộn Xả Metalize M theo cảm biến tiệm cận X4A & Tỷ số truyền Gear_Ratio_M (33/32) *)
Trig_X50 := Sensor_Rev_M AND NOT(Prev_X50);
Prev_X50 := Sensor_Rev_M;
IF Trig_X50 THEN
    Rev_Count_M := Rev_Count_M + 1;
    IF Total_PPR > 0 AND (Curr_Pulse_X2 - Last_Pulse_X2_M) > 0 THEN
        Raw_Dia_M_mm := (DINT_TO_REAL(Curr_Pulse_X2 - Last_Pulse_X2_M) * Dia_X2_Roller_mm * Gear_Ratio_M) / (DINT_TO_REAL(Total_PPR) * Gear_Ratio_X2);
        IF Raw_Dia_M_mm < Core_Dia_M_mm THEN Raw_Dia_M_mm := Core_Dia_M_mm; END_IF;
        IF Raw_Dia_M_mm > Max_Dia_M_mm THEN Raw_Dia_M_mm := Max_Dia_M_mm; END_IF;
        Real_Dia_M_mm := Real_Dia_M_mm + ((Raw_Dia_M_mm - Real_Dia_M_mm) * 0.2);
    END_IF;
    Last_Pulse_X2_M := Curr_Pulse_X2;
END_IF;

(* Đường kính cuộn Xả U theo cảm biến tiệm cận X4B *)
Trig_X51 := Sensor_Rev_U AND NOT(Prev_X51);
Prev_X51 := Sensor_Rev_U;
IF Trig_X51 THEN
    Rev_Count_U := Rev_Count_U + 1;
    IF Total_PPR > 0 AND (Curr_Pulse_X2 - Last_Pulse_X2_U) > 0 THEN
        Raw_Dia_U_mm := (DINT_TO_REAL(Curr_Pulse_X2 - Last_Pulse_X2_U) * Dia_X2_Roller_mm) / (DINT_TO_REAL(Total_PPR) * Gear_Ratio_X2);
        IF Raw_Dia_U_mm < Core_Dia_U_mm THEN Raw_Dia_U_mm := Core_Dia_U_mm; END_IF;
        IF Raw_Dia_U_mm > Max_Dia_U_mm THEN Raw_Dia_U_mm := Max_Dia_U_mm; END_IF;
        Real_Dia_U_mm := Real_Dia_U_mm + ((Raw_Dia_U_mm - Real_Dia_U_mm) * 0.2);
    END_IF;
    Last_Pulse_X2_U := Curr_Pulse_X2;
END_IF;

(* ============================================================================ *)
(* 11. STATE MACHINE VẬN HÀNH DÂY CHUYỀN & BÒ CHẬM NỐI MÀNG                     *)
(* ============================================================================ *)
CASE State_Machine OF
    0: (* STATE_STOPPED *)
        IF Cmd_Jog_Crawl AND NOT(Servo_Not_Ready_Fault) THEN
            Target_Line_MPM := Min_Speed_MPM;
            IF Target_Line_MPM <= 0.0 THEN Target_Line_MPM := 2.0; END_IF;
        ELSE
            Current_Line_MPM := 0.0;
            Target_Line_MPM  := 0.0;
        END_IF;

        IF Cmd_Start AND NOT(Servo_Not_Ready_Fault) THEN
            State_Machine   := 1;
            HMI_PID_Enable  := TRUE;
            HMI_Start       := FALSE;
            IF Target_Line_MPM < Min_Speed_MPM THEN Target_Line_MPM := 20.0; END_IF;
        END_IF;

    1: (* STATE_RUNNING *)
        IF Cmd_Stop THEN
            State_Machine := 0;
            HMI_Stop := FALSE;
        END_IF;
END_CASE;

(* ============================================================================ *)
(* 12. ĐIỀU KHIỂN 5 TRỤC SERVO ON XUẤT RA MODULE QY40 (SLOT 5 - Y50..Y54)        *)
(* ============================================================================ *)
Servo_ON_T  := (State_Machine = 1) OR HMI_Test_T;
Servo_ON_X1 := (State_Machine = 1) OR HMI_Test_X1;
Servo_ON_X2 := (State_Machine = 1) OR HMI_Test_X2;
Servo_ON_Ms := (State_Machine = 1) OR HMI_Test_Ms;
Servo_ON_S  := (State_Machine = 1) OR HMI_Test_S;

Y50 := Servo_ON_T;  (* Servo ON Trục Thu T *)
Y51 := Servo_ON_X1; (* Servo ON Trục Kéo X1 *)
Y52 := Servo_ON_X2; (* Servo ON Trục Master X2 *)
Y53 := Servo_ON_Ms; (* Servo ON Trục Ghép Ms *)
Y54 := Servo_ON_S;  (* Servo ON Trục Dầu S *)

DO_Pen1 := Pen1_State;
DO_Pen2 := Pen2_State;
Y55 := DO_Pen1;
Y56 := DO_Pen2;

DO_Alarm_Horn      := Servo_Not_Ready_Fault;
Tower_Light_Green  := (State_Machine = 1);
Tower_Light_Yellow := (State_Machine = 0) AND (Cmd_Jog_Crawl OR NOT(Servo_Not_Ready_Fault));
Tower_Light_Red    := Servo_Not_Ready_Fault;

Y57 := DO_Alarm_Horn;
Y58 := Tower_Light_Green;
Y59 := Tower_Light_Yellow;
Y5A := Tower_Light_Red;

(* ============================================================================ *)
(* 13. TÍNH CÔN LỰC TAPER TENSION CUỘN THU T (FLOAT)                            *)
(* ============================================================================ *)
IF (Max_Dia_T_mm - Core_Dia_T_mm) > 0.0 AND Taper_Percent_T > 0.0 THEN
    Effective_SP_T := SP_Tension_T - (((Real_Dia_T_mm - Core_Dia_T_mm) * SP_Tension_T * (Taper_Percent_T / 100.0)) / (Max_Dia_T_mm - Core_Dia_T_mm));
ELSE
    Effective_SP_T := SP_Tension_T;
END_IF;
IF Effective_SP_T < 0.0 THEN Effective_SP_T := 0.0; END_IF;

(* Tốc độ đặt Setpoint đồng bộ Master X2 (0..16000) *)
Base_Speed_X2 := (Current_Line_MPM * 16000.0) / Max_Speed_MPM;

SP_Speed_X2 := Base_Speed_X2;
SP_Speed_X1 := (Base_Speed_X2 * Speed_Ratio_X1) + Speed_Offset_X1;
SP_Speed_Ms := (((Base_Speed_X2 * Dia_Ms_Roller_mm) / Dia_X2_Roller_mm) * Speed_Ratio_Ms) + Speed_Offset_Ms;
SP_Speed_S  := (Base_Speed_X2 * Speed_Ratio_S) + Speed_Offset_S;
SP_Speed_T  := ((Base_Speed_X2 * Real_Dia_T_mm) / Core_Dia_T_mm) * Speed_Ratio_T;

(* ============================================================================ *)
(* 14. BỘ CHUYỂN MẠCH INDEX-REGISTER CHO HMI CHỈNH PID, CALIB VÀ ZERO ĐA TRỤC   *)
(* ============================================================================ *)
IF HMI_Axis_Select <= 0 OR HMI_Axis_Select > 7 THEN
    HMI_Axis_Select := 1;
END_IF;

IF HMI_Cmd_Save_PID THEN
    CASE HMI_Axis_Select OF
        1: Kp_T := HMI_Disp_Kp; Ki_T := HMI_Disp_Ki; Kd_T := HMI_Disp_Kd; Calib_Gain_T := HMI_Disp_Calib_Gain; Zero_Offset_T := HMI_Disp_Zero_Offset;
        2: Kp_X1 := HMI_Disp_Kp; Ki_X1 := HMI_Disp_Ki; Kd_X1 := HMI_Disp_Kd; Calib_Gain_X1 := HMI_Disp_Calib_Gain; Zero_Offset_X1 := HMI_Disp_Zero_Offset;
        3: Kp_X2 := HMI_Disp_Kp; Ki_X2 := HMI_Disp_Ki; Kd_X2 := HMI_Disp_Kd;
        4: Kp_Ms := HMI_Disp_Kp; Ki_Ms := HMI_Disp_Ki; Kd_Ms := HMI_Disp_Kd;
        5: Kp_S := HMI_Disp_Kp; Ki_S := HMI_Disp_Ki; Kd_S := HMI_Disp_Kd;
        6: Kp_M := HMI_Disp_Kp; Ki_M := HMI_Disp_Ki; Kd_M := HMI_Disp_Kd; Calib_Gain_M := HMI_Disp_Calib_Gain; Zero_Offset_M := HMI_Disp_Zero_Offset;
        7: Kp_U := HMI_Disp_Kp; Ki_U := HMI_Disp_Ki; Kd_U := HMI_Disp_Kd; Calib_Gain_U := HMI_Disp_Calib_Gain; Zero_Offset_U := HMI_Disp_Zero_Offset;
    END_CASE;
    HMI_Cmd_Save_PID := FALSE;
ELSE
    CASE HMI_Axis_Select OF
        1: HMI_Disp_Kp := Kp_T; HMI_Disp_Ki := Ki_T; HMI_Disp_Kd := Kd_T; HMI_Disp_Calib_Gain := Calib_Gain_T; HMI_Disp_Zero_Offset := Zero_Offset_T;
        2: HMI_Disp_Kp := Kp_X1; HMI_Disp_Ki := Ki_X1; HMI_Disp_Kd := Kd_X1; HMI_Disp_Calib_Gain := Calib_Gain_X1; HMI_Disp_Zero_Offset := Zero_Offset_X1;
        3: HMI_Disp_Kp := Kp_X2; HMI_Disp_Ki := Ki_X2; HMI_Disp_Kd := Kd_X2; HMI_Disp_Calib_Gain := 1.0; HMI_Disp_Zero_Offset := 0.0;
        4: HMI_Disp_Kp := Kp_Ms; HMI_Disp_Ki := Ki_Ms; HMI_Disp_Kd := Kd_Ms; HMI_Disp_Calib_Gain := 1.0; HMI_Disp_Zero_Offset := 0.0;
        5: HMI_Disp_Kp := Kp_S; HMI_Disp_Ki := Ki_S; HMI_Disp_Kd := Kd_S; HMI_Disp_Calib_Gain := 1.0; HMI_Disp_Zero_Offset := 0.0;
        6: HMI_Disp_Kp := Kp_M; HMI_Disp_Ki := Ki_M; HMI_Disp_Kd := Kd_M; HMI_Disp_Calib_Gain := Calib_Gain_M; HMI_Disp_Zero_Offset := Zero_Offset_M;
        7: HMI_Disp_Kp := Kp_U; HMI_Disp_Ki := Ki_U; HMI_Disp_Kd := Kd_U; HMI_Disp_Calib_Gain := Calib_Gain_U; HMI_Disp_Zero_Offset := Zero_Offset_U;
    END_CASE;
END_IF;

IF Calib_Set_T OR (HMI_Cmd_Calib_Set AND HMI_Axis_Select = 1) THEN
    Calib_Gain_T := HMI_Disp_Calib_Gain; Calib_Set_T := FALSE;
END_IF;
IF Calib_Set_X1 OR (HMI_Cmd_Calib_Set AND HMI_Axis_Select = 2) THEN
    Calib_Gain_X1 := HMI_Disp_Calib_Gain; Calib_Set_X1 := FALSE;
END_IF;
IF Calib_Set_M OR (HMI_Cmd_Calib_Set AND HMI_Axis_Select = 6) THEN
    Calib_Gain_M := HMI_Disp_Calib_Gain; Calib_Set_M := FALSE;
END_IF;
IF Calib_Set_U OR (HMI_Cmd_Calib_Set AND HMI_Axis_Select = 7) THEN
    Calib_Gain_U := HMI_Disp_Calib_Gain; Calib_Set_U := FALSE;
END_IF;
IF HMI_Cmd_Calib_Set THEN
    HMI_Cmd_Calib_Set := FALSE;
END_IF;

(* ============================================================================ *)
(* 15. TÍNH TỐC ĐỘ RPM/MPM VÀ GỌI RUN CÁC KHỐI PID THEO NHỊP 10MS TỪ SM409      *)
(* ============================================================================ *)
Trig_PID_10ms := SM409 AND NOT(Prev_SM409);
Prev_SM409 := SM409;

IF Trig_PID_10ms THEN
    (* 15.1. Tính Delta xung trong chu kỳ 10ms *)
    Delta_T   := ABS(Curr_Pulse_T  - Prev_Pulse_T);
    Delta_X1  := ABS(Curr_Pulse_X1 - Prev_Pulse_X1);
    Delta_X2  := ABS(Curr_Pulse_X2 - Prev_Pulse_X2);
    Delta_Ms  := ABS(Curr_Pulse_Ms - Prev_Pulse_Ms);

    Prev_Pulse_T  := Curr_Pulse_T;
    Prev_Pulse_X1 := Curr_Pulse_X1;
    Prev_Pulse_X2 := Curr_Pulse_X2;
    Prev_Pulse_Ms := Curr_Pulse_Ms;

    Total_PPR := PPR_Encoder * 4; (* 2000 x 4 = 8000 *)

    (* 15.2. TÍNH TOÁN TỐC ĐỘ RPM THÔ (Chu kỳ 10ms: Delta * 6000.0 / Total_PPR) *)
    IF Total_PPR > 0 THEN
        Raw_RPM_T  := (DINT_TO_REAL(Delta_T)  * 6000.0) / DINT_TO_REAL(Total_PPR);
        Raw_RPM_X1 := (DINT_TO_REAL(Delta_X1) * 6000.0) / DINT_TO_REAL(Total_PPR);
        Raw_RPM_X2 := (DINT_TO_REAL(Delta_X2) * 6000.0) / DINT_TO_REAL(Total_PPR);
        Raw_RPM_Ms := (DINT_TO_REAL(Delta_Ms) * 6000.0) / DINT_TO_REAL(Total_PPR);
    END_IF;

    (* TÍNH TỐC ĐỘ TRỤC S THÔ TỪ ANALOG OUT SERVO (Q68ADV CH5 - U0\G5: 0..16000 = 0..Max_RPM_S) *)
    Raw_Analog_S := INT_TO_REAL(ADC_CH5_Raw);
    IF Raw_Analog_S < 0.0 THEN Raw_Analog_S := 0.0; ELSIF Raw_Analog_S > 16000.0 THEN Raw_Analog_S := 16000.0; END_IF;

    IF Max_RPM_S > 0.0 THEN
        Raw_RPM_S := (Raw_Analog_S * Max_RPM_S) / 16000.0;
    ELSE
        Raw_RPM_S := 0.0;
    END_IF;

    (* 15.3. BỘ LỌC TRUNG BÌNH TRƯỢT 4 MẪU (MOVING AVERAGE GIỐNG MODULE ADC Q68ADV) *)
    RPM_T  := (Raw_RPM_T  + Buf_RPM_T_1  + Buf_RPM_T_2  + Buf_RPM_T_3)  / 4.0;
    RPM_X1 := (Raw_RPM_X1 + Buf_RPM_X1_1 + Buf_RPM_X1_2 + Buf_RPM_X1_3) / 4.0;
    RPM_X2 := (Raw_RPM_X2 + Buf_RPM_X2_1 + Buf_RPM_X2_2 + Buf_RPM_X2_3) / 4.0;
    RPM_Ms := (Raw_RPM_Ms + Buf_RPM_Ms_1 + Buf_RPM_Ms_2 + Buf_RPM_Ms_3) / 4.0;
    RPM_S  := (Raw_RPM_S  + Buf_RPM_S_1  + Buf_RPM_S_2  + Buf_RPM_S_3)  / 4.0;

    (* Dịch chuyển bộ nhớ đệm mẫu trượt *)
    Buf_RPM_T_3  := Buf_RPM_T_2;   Buf_RPM_T_2  := Buf_RPM_T_1;   Buf_RPM_T_1  := Raw_RPM_T;
    Buf_RPM_X1_3 := Buf_RPM_X1_2;  Buf_RPM_X1_2 := Buf_RPM_X1_1;  Buf_RPM_X1_1 := Raw_RPM_X1;
    Buf_RPM_X2_3 := Buf_RPM_X2_2;  Buf_RPM_X2_2 := Buf_RPM_X2_1;  Buf_RPM_X2_1 := Raw_RPM_X2;
    Buf_RPM_Ms_3 := Buf_RPM_Ms_2;  Buf_RPM_Ms_2 := Buf_RPM_Ms_1;  Buf_RPM_Ms_1 := Raw_RPM_Ms;
    Buf_RPM_S_3  := Buf_RPM_S_2;   Buf_RPM_S_2  := Buf_RPM_S_1;   Buf_RPM_S_1  := Raw_RPM_S;

    (* 15.4. TÍNH VẬN TỐC DÂY MPM (PI = 3.1415) *)
    IF Gear_Ratio_T > 0.0 THEN
        MPM_T  := (RPM_T  * 3.1415 * Real_Dia_T_mm)    / (1000.0 * Gear_Ratio_T);
    END_IF;
    IF Gear_Ratio_X1 > 0.0 THEN
        MPM_X1 := (RPM_X1 * 3.1415 * Dia_X1_Roller_mm) / (1000.0 * Gear_Ratio_X1);
    END_IF;
    IF Gear_Ratio_X2 > 0.0 THEN
        MPM_X2 := (RPM_X2 * 3.1415 * Dia_X2_Roller_mm) / (1000.0 * Gear_Ratio_X2);
    END_IF;
    IF Gear_Ratio_Ms > 0.0 THEN
        MPM_Ms := (RPM_Ms * 3.1415 * Dia_Ms_Roller_mm) / (1000.0 * Gear_Ratio_Ms);
    END_IF;
    IF Gear_Ratio_S > 0.0 THEN
        MPM_S  := (RPM_S  * 3.1415 * Dia_S_Roller_mm)  / (1000.0 * Gear_Ratio_S);
    END_IF;

    (* 15.5. GÁN BIẾN FEEDBACK CHO CÁC VÒNG PID TỐC ĐỘ (0..16000 DAC) *)
    IF Max_RPM_X2 > 0.0 THEN
        Feedback_Speed_X2 := (RPM_X2 * 16000.0) / Max_RPM_X2;
    END_IF;
    IF Max_RPM_Ms > 0.0 THEN
        Feedback_Speed_Ms := (RPM_Ms * 16000.0) / Max_RPM_Ms;
    END_IF;
    Feedback_Speed_S := Raw_Analog_S;

    (* 15.6. GỌI CÁC KHỐI PID *)
    (* PID Tốc độ Trục chính Master X2 *)
    pid_X2(
        Enable      := (HMI_PID_Enable AND State_Machine = 1) OR (HMI_Cmd_AutoTune AND HMI_Axis_Select = 3),
        Setpoint    := SP_Speed_X2,
        Feedback    := Feedback_Speed_X2,
        Kp          := Kp_X2, Ki := Ki_X2, Kd := Kd_X2,
        AT_Enable   := (HMI_Cmd_AutoTune AND HMI_Axis_Select = 3)
    );
    PID_Out_X2 := pid_X2.PID_Output;

    (* PID Tốc độ Trục Ghép Ms *)
    pid_Ms(
        Enable      := (HMI_PID_Enable AND State_Machine = 1) OR (HMI_Cmd_AutoTune AND HMI_Axis_Select = 4),
        Setpoint    := SP_Speed_Ms,
        Feedback    := Feedback_Speed_Ms,
        Kp          := Kp_Ms, Ki := Ki_Ms, Kd := Kd_Ms,
        AT_Enable   := (HMI_Cmd_AutoTune AND HMI_Axis_Select = 4)
    );
    PID_Out_Ms := pid_Ms.PID_Output;

    (* PID Tốc độ Trục Tráng Dầu S (Feedback từ Analog Out Servo đấu vào Q68ADV CH5) *)
    pid_S(
        Enable      := (HMI_PID_Enable AND State_Machine = 1) OR (HMI_Cmd_AutoTune AND HMI_Axis_Select = 5),
        Setpoint    := SP_Speed_S,
        Feedback    := Feedback_Speed_S,
        Kp          := Kp_S, Ki := Ki_S, Kd := Kd_S,
        AT_Enable   := (HMI_Cmd_AutoTune AND HMI_Axis_Select = 5)
    );
    PID_Out_S := pid_S.PID_Output;

    (* PID Lực căng Loadcell Trục Kéo Giấy X1 *)
    pid_X1(
        Enable      := (HMI_PID_Enable AND State_Machine = 1) OR (HMI_Cmd_AutoTune AND HMI_Axis_Select = 2),
        Setpoint    := SP_Tension_X1,
        Feedback    := Weight_Net_X1,
        Kp          := Kp_X1, Ki := Ki_X1, Kd := Kd_X1,
        AT_Enable   := (HMI_Cmd_AutoTune AND HMI_Axis_Select = 2)
    );
    PID_Out_X1 := pid_X1.PID_Output;

    (* PID Lực căng Loadcell Cuộn Thu T *)
    pid_T(
        Enable      := (HMI_PID_Enable AND State_Machine = 1) OR (HMI_Cmd_AutoTune AND HMI_Axis_Select = 1),
        Setpoint    := Effective_SP_T,
        Feedback    := Weight_Net_T,
        Kp          := Kp_T, Ki := Ki_T, Kd := Kd_T,
        AT_Enable   := (HMI_Cmd_AutoTune AND HMI_Axis_Select = 1)
    );
    PID_Out_T := pid_T.PID_Output;

    (* PID Lực căng Thắng Từ Xả M *)
    pid_M(
        Enable      := (HMI_PID_Enable AND State_Machine = 1) OR (HMI_Cmd_AutoTune AND HMI_Axis_Select = 6),
        Setpoint    := SP_Tension_M,
        Feedback    := Weight_Net_M,
        Kp          := Kp_M, Ki := Ki_M, Kd := Kd_M,
        AT_Enable   := (HMI_Cmd_AutoTune AND HMI_Axis_Select = 6)
    );
    PID_Out_M := pid_M.PID_Output;

    (* PID Lực căng Trục Xả Metalize U *)
    pid_U(
        Enable      := (HMI_PID_Enable AND State_Machine = 1) OR (HMI_Cmd_AutoTune AND HMI_Axis_Select = 7),
        Setpoint    := SP_Tension_U,
        Feedback    := Weight_Net_U,
        Kp          := Kp_U, Ki := Ki_U, Kd := Kd_U,
        AT_Enable   := (HMI_Cmd_AutoTune AND HMI_Axis_Select = 7)
    );
    PID_Out_U := pid_U.PID_Output;

    (* TỰ ĐỘNG CẬP NHẬT KẾT QUẢ KHI AUTO-TUNE HOÀN THÀNH *)
    IF pid_X2.AT_Done THEN
        Kp_X2 := pid_X2.Tuned_Kp; Ki_X2 := pid_X2.Tuned_Ki; Kd_X2 := pid_X2.Tuned_Kd;
        HMI_Disp_Kp := Kp_X2; HMI_Disp_Ki := Ki_X2; HMI_Disp_Kd := Kd_X2;
    ELSIF pid_Ms.AT_Done THEN
        Kp_Ms := pid_Ms.Tuned_Kp; Ki_Ms := pid_Ms.Tuned_Ki; Kd_Ms := pid_Ms.Tuned_Kd;
        HMI_Disp_Kp := Kp_Ms; HMI_Disp_Ki := Ki_Ms; HMI_Disp_Kd := Kd_Ms;
    ELSIF pid_S.AT_Done THEN
        Kp_S := pid_S.Tuned_Kp; Ki_S := pid_S.Tuned_Ki; Kd_S := pid_S.Tuned_Kd;
        HMI_Disp_Kp := Kp_S; HMI_Disp_Ki := Ki_S; HMI_Disp_Kd := Kd_S;
    ELSIF pid_X1.AT_Done THEN
        Kp_X1 := pid_X1.Tuned_Kp; Ki_X1 := pid_X1.Tuned_Ki; Kd_X1 := pid_X1.Tuned_Kd;
        HMI_Disp_Kp := Kp_X1; HMI_Disp_Ki := Ki_X1; HMI_Disp_Kd := Kd_X1;
    ELSIF pid_T.AT_Done THEN
        Kp_T := pid_T.Tuned_Kp; Ki_T := pid_T.Tuned_Ki; Kd_T := pid_T.Tuned_Kd;
        HMI_Disp_Kp := Kp_T; HMI_Disp_Ki := Ki_T; HMI_Disp_Kd := Kd_T;
    ELSIF pid_M.AT_Done THEN
        Kp_M := pid_M.Tuned_Kp; Ki_M := pid_M.Tuned_Ki; Kd_M := pid_M.Tuned_Kd;
        HMI_Disp_Kp := Kp_M; HMI_Disp_Ki := Ki_M; HMI_Disp_Kd := Kd_M;
    ELSIF pid_U.AT_Done THEN
        Kp_U := pid_U.Tuned_Kp; Ki_U := pid_U.Tuned_Ki; Kd_U := pid_U.Tuned_Kd;
        HMI_Disp_Kp := Kp_U; HMI_Disp_Ki := Ki_U; HMI_Disp_Kd := Kd_U;
    END_IF;

    IF pid_X2.AT_Done OR pid_Ms.AT_Done OR pid_S.AT_Done OR pid_X1.AT_Done OR pid_T.AT_Done OR pid_M.AT_Done OR pid_U.AT_Done THEN
        HMI_Cmd_AutoTune   := FALSE;
        HMI_Status_AT_Done := TRUE;
    END_IF;
    
    HMI_Status_AT_Busy := pid_T.AT_Busy OR pid_X1.AT_Busy OR pid_X2.AT_Busy OR pid_Ms.AT_Busy OR pid_S.AT_Busy OR pid_M.AT_Busy OR pid_U.AT_Busy;
END_IF;

(* ============================================================================ *)
(* 16. TÍNH TOÁN XUẤT ÁP TỐC ĐỘ VÀ TORQUE CHO TỪNG TRỤC (FLOAT)                  *)
(* ============================================================================ *)
IF State_Machine = 0 THEN
    IF HMI_Test_X2 THEN Calc_Speed_X2 := Test_Speed_X2; ELSE Calc_Speed_X2 := 0.0; END_IF;
    IF HMI_Test_X1 THEN Calc_Speed_X1 := Test_Speed_X1; ELSE Calc_Speed_X1 := 0.0; END_IF;
    IF HMI_Test_Ms THEN Calc_Speed_Ms := Test_Speed_Ms; ELSE Calc_Speed_Ms := 0.0; END_IF;
    IF HMI_Test_S  THEN Calc_Speed_S  := Test_Speed_S;  ELSE Calc_Speed_S  := 0.0; END_IF;

    IF HMI_Test_T THEN
        Calc_Speed_T  := Test_Speed_T;
        Calc_Torque_T := Test_Torque_T;
    ELSE
        Calc_Speed_T  := 0.0;
        Calc_Torque_T := 0.0;
    END_IF;

    IF HMI_Test_M THEN
        Calc_Torque_M := Test_Torque_M;
    ELSIF Hold_Torque_Stop_M THEN
        Calc_Torque_M := (Base_Torque_M * 80.0);
    ELSE
        Calc_Torque_M := 0.0;
    END_IF;

    IF HMI_Test_U THEN
        Calc_Speed_U := Test_Speed_U;
    ELSIF Hold_Torque_Stop_U THEN
        Calc_Speed_U := (Init_Holding_Torque_U * 80.0);
    ELSE
        Calc_Speed_U := 0.0;
    END_IF;

ELSE
    Calc_Speed_X2 := SP_Speed_X2 + PID_Out_X2;
    Calc_Speed_X1 := SP_Speed_X1 + PID_Out_X1;
    Calc_Speed_Ms := SP_Speed_Ms + PID_Out_Ms;
    Calc_Speed_S  := SP_Speed_S  + PID_Out_S;
    Calc_Speed_T  := SP_Speed_T;
    Calc_Torque_T := (Effective_SP_T * 160.0) + PID_Out_T;

    (* Xả U: Giới hạn ngõ ra max 5V (tương đương 0..8000 trên dải 0..10V) *)
    IF Real_Dia_U_mm > 0.0 THEN
        Calc_Speed_U := (((Calc_Speed_X2 * Max_Dia_U_mm) / Real_Dia_U_mm) * 0.5) + PID_Out_U;
    ELSE
        Calc_Speed_U := (Calc_Speed_X2 * 0.5) + PID_Out_U;
    END_IF;

    IF Rev_Count_M <= 5 THEN
        Base_Torque_M := Init_Holding_Torque_M;
    ELSIF (Max_Dia_M_mm - Core_Dia_M_mm) > 0.0 THEN
        Base_Torque_M := Min_Torque_M + (((Max_Torque_M - Min_Torque_M) * (Real_Dia_M_mm - Core_Dia_M_mm)) / (Max_Dia_M_mm - Core_Dia_M_mm));
    ELSE
        Base_Torque_M := Min_Torque_M;
    END_IF;
    (* Thắng Từ M: Giới hạn ngõ ra max 5V (0..100% ứng với 0..8000) *)
    Calc_Torque_M := (Base_Torque_M * 80.0) + PID_Out_M;
END_IF;

(* Khống chế biên an toàn ngõ ra Analog: Các trục Servo xuất 0..16000 (0..10V), riêng Thắng M và Xả U xuất 0..8000 (0..5V) *)
IF Calc_Speed_T  < 0.0 THEN Calc_Speed_T  := 0.0; ELSIF Calc_Speed_T  > 16000.0 THEN Calc_Speed_T  := 16000.0; END_IF;
IF Calc_Torque_T < 0.0 THEN Calc_Torque_T := 0.0; ELSIF Calc_Torque_T > 16000.0 THEN Calc_Torque_T := 16000.0; END_IF;
IF Calc_Speed_X1 < 0.0 THEN Calc_Speed_X1 := 0.0; ELSIF Calc_Speed_X1 > 16000.0 THEN Calc_Speed_X1 := 16000.0; END_IF;
IF Calc_Speed_X2 < 0.0 THEN Calc_Speed_X2 := 0.0; ELSIF Calc_Speed_X2 > 16000.0 THEN Calc_Speed_X2 := 16000.0; END_IF;
IF Calc_Speed_Ms < 0.0 THEN Calc_Speed_Ms := 0.0; ELSIF Calc_Speed_Ms > 16000.0 THEN Calc_Speed_Ms := 16000.0; END_IF;
IF Calc_Torque_M < 0.0 THEN Calc_Torque_M := 0.0; ELSIF Calc_Torque_M > 8000.0  THEN Calc_Torque_M := 8000.0;  END_IF;
IF Calc_Speed_S  < 0.0 THEN Calc_Speed_S  := 0.0; ELSIF Calc_Speed_S  > 16000.0 THEN Calc_Speed_S  := 16000.0; END_IF;
IF Calc_Speed_U  < 0.0 THEN Calc_Speed_U  := 0.0; ELSIF Calc_Speed_U  > 8000.0  THEN Calc_Speed_U  := 8000.0;  END_IF;

(* ============================================================================ *)
(* 17. XUẤT TRỰC TIẾP RA BUFFER MEMORY MODULE Q68DAV (SLOT 1 - U1\G1..U1\G8)     *)
(* ============================================================================ *)
U1\G1 := REAL_TO_INT(Calc_Speed_T);  (* CH1: Speed Thu T (0..16000) *)
U1\G2 := REAL_TO_INT(Calc_Torque_T); (* CH2: Torque Thu T (0..16000) *)
U1\G3 := REAL_TO_INT(Calc_Speed_X1); (* CH3: Speed Kéo X1 (0..16000) *)
U1\G4 := REAL_TO_INT(Calc_Speed_X2); (* CH4: Speed Master X2 (0..16000) *)
U1\G5 := REAL_TO_INT(Calc_Speed_Ms); (* CH5: Speed Ghép Ms (0..16000) *)
U1\G6 := REAL_TO_INT(Calc_Torque_M); (* CH6: Torque Thắng M (0..16000) *)
U1\G7 := REAL_TO_INT(Calc_Speed_S);  (* CH7: Speed Tráng Dầu S (0..16000) *)
U1\G8 := REAL_TO_INT(Calc_Speed_U);  (* CH8: Speed Xả U (0..16000) *)

D510 := INT_TO_WORD(U1\G1);
D511 := INT_TO_WORD(U1\G2);
D512 := INT_TO_WORD(U1\G3);
D513 := INT_TO_WORD(U1\G4);
D514 := INT_TO_WORD(U1\G5);
D515 := INT_TO_WORD(U1\G6);
D516 := INT_TO_WORD(U1\G7);
D517 := INT_TO_WORD(U1\G8);

(* ============================================================================ *)
(* 18. TỰ ĐỘNG BÁO GIẢM TỐC VÀ DỪNG MÁY KHI ĐẠT CHIỀU DÀI MÉT CÀI ĐẶT           *)
(* ============================================================================ *)
IF Set_Target_Length > 0.0 AND State_Machine = 1 THEN
    IF Total_Length_Meters >= Set_Target_Length THEN
        State_Machine    := 0;
        Target_Line_MPM  := 0.0;
        Current_Line_MPM := 0.0;
    ELSIF Decel_Distance_Meters > 0.0 AND Total_Length_Meters >= (Set_Target_Length - Decel_Distance_Meters) THEN
        IF Target_Line_MPM > Min_Speed_MPM THEN Target_Line_MPM := Min_Speed_MPM; END_IF;
    END_IF;
END_IF;

Auto_Decel_Flag := (Set_Target_Length > 0.0) AND (State_Machine = 1) AND (Decel_Distance_Meters > 0.0) AND (Total_Length_Meters >= (Set_Target_Length - Decel_Distance_Meters)) AND (Total_Length_Meters < Set_Target_Length);

(* ============================================================================ *)
(* 19. CẬP NHẬT MÃ TRẠNG THÁI HIỂN THỊ TIẾNG VIỆT TRÊN HMI CHO CÔNG NHÂN        *)
(* ============================================================================ *)
IF Servo_Not_Ready_Fault THEN
    HMI_Status_Text_Code := 1; (* Báo lỗi 5 Servo *)
ELSIF State_Machine = 1 THEN
    HMI_Status_Text_Code := 2; (* Đang chạy tự động *)
ELSIF Cmd_Jog_Crawl THEN
    HMI_Status_Text_Code := 3; (* Đang bò chậm nối màng *)
ELSIF Auto_Decel_Flag OR (Set_Target_Length > 0.0 AND Total_Length_Meters >= Set_Target_Length) THEN
    HMI_Status_Text_Code := 4; (* Đã hoàn thành đơn hàng *)
ELSE
    HMI_Status_Text_Code := 0; (* Máy dừng - Sẵn sàng chạy *)
END_IF;
END_PROGRAM

FUNCTION_BLOCK FB_TENSION_PID
VAR_INPUT
  Enable : BOOL;
  Reset : BOOL;
  Setpoint : REAL;
  Feedback : REAL;
  Kp : REAL;
  Ki : REAL;
  Kd : REAL;
  Deadband : REAL;
  Out_Min : REAL;
  Out_Max : REAL;
  AT_Enable : BOOL;
  AT_Step : REAL;
END_VAR
VAR_OUTPUT
  PID_Output : REAL;
  Error : REAL;
  AT_Done : BOOL;
  AT_Busy : BOOL;
  Tuned_Kp : REAL;
  Tuned_Ki : REAL;
  Tuned_Kd : REAL;
END_VAR
VAR
  Error_Prev : REAL;
  I_Term : REAL;
  P_Term : REAL;
  D_Term : REAL;
  AT_State : INT;
  AT_Cycle_Count : INT;
  AT_Timer_10ms : DINT;
  AT_Period_Tu : REAL;
  AT_Ku : REAL;
  AT_PV_Max : REAL;
  AT_PV_Min : REAL;
  AT_Base_Out : REAL;
  AT_Relay_State : BOOL;
  Test_Step : REAL;
END_VAR
(* ============================================================================ *)
(* FUNCTION BLOCK: FB_TENSION_PID (ĐIỀU KHIỂN PID & AUTO-TUNING TỰ ĐỘNG TÌM THÔNG SỐ) *)
(* PHƯƠNG PHÁP AUTO-TUNING: RELAY FEEDBACK LIMIT-CYCLE (ZIEGLER-NICHOLS CẢI TIẾN) *)
(* ============================================================================ *)

IF NOT Enable THEN
    PID_Output := 0.0;
    I_Term     := 0.0;
    Error_Prev := 0.0;
    AT_Busy    := FALSE;
    AT_State   := 0;
    RETURN;
END_IF;

IF Reset THEN
    I_Term     := 0.0;
    Error_Prev := 0.0;
    PID_Output := 0.0;
    AT_Busy    := FALSE;
    AT_State   := 0;
    AT_Done    := FALSE;
    RETURN;
END_IF;

(* ============================================================================ *)
(* 1. CHẾ ĐỘ AUTO-TUNING (DÒ THÔNG SỐ TỰ ĐỘNG BẰNG RELAY LIMIT-CYCLE)           *)
(* ============================================================================ *)
IF AT_Enable THEN
    AT_Busy := TRUE;
    AT_Done := FALSE;
    
    (* Sử dụng biến nội bộ Test_Step để không ghi đè vào VAR_INPUT AT_Step *)
    IF AT_Step > 0.0 THEN
        Test_Step := AT_Step;
    ELSE
        Test_Step := 800.0; (* Mặc định 800 đơn vị DAC ~ 5% của 16000 *)
    END_IF;

    CASE AT_State OF
        0: (* KHỞI TẠO BƯỚC TEST *)
            AT_Base_Out     := PID_Output;
            AT_PV_Max       := Feedback;
            AT_PV_Min       := Feedback;
            AT_Cycle_Count  := 0;
            AT_Timer_10ms   := 0;
            AT_Relay_State  := TRUE;
            AT_State        := 1;

        1: (* THỰC THI DAO ĐỘNG BẬT/TẮT RELAY QUA SETPOINT *)
            AT_Timer_10ms := AT_Timer_10ms + 1;

            (* Theo dõi giá trị đỉnh/đáy của Feedback *)
            IF Feedback > AT_PV_Max THEN AT_PV_Max := Feedback; END_IF;
            IF Feedback < AT_PV_Min THEN AT_PV_Min := Feedback; END_IF;

            (* Điều khiển Relay đảo trạng thái khi vượt qua Setpoint *)
            IF AT_Relay_State THEN
                PID_Output := AT_Base_Out + Test_Step;
                IF Feedback >= Setpoint THEN
                    AT_Relay_State := FALSE;
                END_IF;
            ELSE
                PID_Output := AT_Base_Out - Test_Step;
                IF Feedback < Setpoint THEN
                    AT_Relay_State := TRUE;
                    AT_Cycle_Count := AT_Cycle_Count + 1; (* Đếm xong 1 chu kỳ hoàn chỉnh *)
                END_IF;
            END_IF;

            (* Khi hoàn thành đủ 3 chu kỳ dao động chuẩn *)
            IF AT_Cycle_Count >= 3 THEN
                AT_State := 2;
            END_IF;

        2: (* TÍNH TOÁN BỘ THÔNG SỐ TUNED_KP, TUNED_KI, TUNED_KD *)
            (* Chu kỳ dao động riêng Tu (giây) = tổng thời gian 3 chu kỳ / 3 *)
            IF AT_Timer_10ms > 0 THEN
                AT_Period_Tu := (DINT_TO_REAL(AT_Timer_10ms) * 0.01) / 3.0;
            ELSE
                AT_Period_Tu := 1.0;
            END_IF;

            (* Biên độ dao động đáp ứng A = (PV_Max - PV_Min) / 2 *)
            IF (AT_PV_Max - AT_PV_Min) > 0.1 THEN
                (* Độ khuếch đại tới hạn Ku = 4 * Test_Step / (PI * A) *)
                AT_Ku := (4.0 * Test_Step) / (3.141593 * ((AT_PV_Max - AT_PV_Min) / 2.0));
            ELSE
                AT_Ku := 1.0;
            END_IF;

            (* TÍNH THEO CÔNG THỨC ZIEGLER-NICHOLS CHỐNG VỌT LỐ (NO-OVERSHOOT) *)
            Tuned_Kp := AT_Ku * 0.35;                   (* Kp an toàn êm ái *)
            
            IF AT_Period_Tu > 0.05 THEN
                Tuned_Ki := Tuned_Kp * (0.01 / (AT_Period_Tu * 0.85)); (* Ki cho chu kỳ 10ms *)
                Tuned_Kd := Tuned_Kp * ((AT_Period_Tu * 0.12) / 0.01); (* Kd cho chu kỳ 10ms *)
            ELSE
                Tuned_Ki := Tuned_Kp * 0.05;
                Tuned_Kd := Tuned_Kp * 0.02;
            END_IF;

            (* Khống chế biên an toàn *)
            IF Tuned_Kp < 0.1 THEN Tuned_Kp := 0.1; ELSIF Tuned_Kp > 20.0 THEN Tuned_Kp := 20.0; END_IF;
            IF Tuned_Ki < 0.001 THEN Tuned_Ki := 0.001; ELSIF Tuned_Ki > 5.0 THEN Tuned_Ki := 5.0; END_IF;
            IF Tuned_Kd < 0.0 THEN Tuned_Kd := 0.0; ELSIF Tuned_Kd > 5.0 THEN Tuned_Kd := 5.0; END_IF;

            AT_Busy  := FALSE;
            AT_Done  := TRUE;
            AT_State := 0;
    END_CASE;

    (* Giới hạn biên đầu ra trong lúc test *)
    IF PID_Output > Out_Max THEN PID_Output := Out_Max; END_IF;
    IF PID_Output < Out_Min THEN PID_Output := Out_Min; END_IF;
    RETURN;
END_IF;

(* Khi tắt AT_Enable *)
IF AT_Busy THEN
    AT_Busy  := FALSE;
    AT_State := 0;
END_IF;

(* ============================================================================ *)
(* 2. CHẾ ĐỘ ĐIỀU KHIỂN PID TIÊU CHUẨN (NORMAL RUNNING)                        *)
(* ============================================================================ *)

(* 1. TÍNH ĐỘ LỆCH ERROR E(K) *)
Error := Setpoint - Feedback;

(* 2. BỘ LỌC VÙNG CHẾT DEADBAND *)
IF ABS(Error) <= Deadband THEN
    Error := 0.0;
END_IF;

(* 3. TÍNH THÀNH PHẦN PROPORTIONAL (P) *)
P_Term := Error * Kp;

(* 4. TÍNH THÀNH PHẦN INTEGRAL (I) VỚI CHỐNG BÃO HÒA ANTI-WINDUP *)
I_Term := I_Term + (Error * Ki);

IF Out_Max > Out_Min THEN
    IF I_Term > Out_Max THEN
        I_Term := Out_Max;
    ELSIF I_Term < Out_Min THEN
        I_Term := Out_Min;
    END_IF;
END_IF;

(* 5. TÍNH THÀNH PHẦN DERIVATIVE (D) *)
D_Term := (Error - Error_Prev) * Kd;
Error_Prev := Error;

(* 6. TỔNG HỢP NỔI PID VÀ ÉP BIÊN OUT_MIN..OUT_MAX *)
PID_Output := P_Term + I_Term + D_Term;

IF Out_Max > Out_Min THEN
    IF PID_Output > Out_Max THEN
        PID_Output := Out_Max;
    ELSIF PID_Output < Out_Min THEN
        PID_Output := Out_Min;
    END_IF;
END_IF;
END_FUNCTION_BLOCK

PROGRAM POU_INIT
(* ============================================================================ *)
(* TÊN CHƯƠNG TRÌNH : INIT_PROGRAM (INITIAL EXECUTION POU - KHỞI TẠO HỆ THỐNG)    *)
(* HỆ THỐNG        : MÁY GHÉP MÀNG METALIZE TỰ ĐỘNG - MITSUBISHI Q02U PLC       *)
(* KIỂU DỮ LIỆU    : SỐ THỰC FLOAT / REAL (CHUẨN IEC)                          *)
(* CẤU TRÚC PHẦN CỨNG MỚI (DIRECT BASE RACK - KHÔNG DÙNG CC-LINK):             *)
(*   - SLOT 0 (H00): Q68ADV (8 CH Analog Input: Loadcell T, X1, M, U & Analog S)*)
(*   - SLOT 1 (H10): Q68DAV (8 CH Analog Output: Speed/Torque T, X1, X2, Ms, S, M, U) *)
(*   - SLOT 2 (H20): QD62D  (2 CH High Speed Counter: Trục T & Trục X1)        *)
(*   - SLOT 3 (H30): QD62D  (2 CH High Speed Counter: Trục X2 & Trục Ms)       *)
(*   - SLOT 4 (H40): QX40   (16 CH Digital Input: X40..X4F)                    *)
(*   - SLOT 5 (H50): QY40   (16 CH Digital Output: Y50..Y5F)                   *)
(*   - SLOT 6 (H60): QJ71C24N (RS232/RS485 Communication)                      *)
(* ============================================================================ *)

(* ---------------------------------------------------------------------------- *)
(* 1. KHỞI TẠO TỐC ĐỘ TỐI ĐA MOTOR (RPM - REAL)                                *)
(* ---------------------------------------------------------------------------- *)
IF Max_RPM_X2 <= 0.0 THEN Max_RPM_X2 := 1000.0; END_IF; (* Trục Master X2: Max 1000 RPM *)
IF Max_RPM_X1 <= 0.0 THEN Max_RPM_X1 := 1000.0; END_IF; (* Trục Kéo X1:    Max 1000 RPM *)
IF Max_RPM_Ms <= 0.0 THEN Max_RPM_Ms := 3000.0; END_IF; (* Trục Ghép Ms:   Max 3000 RPM *)
IF Max_RPM_S  <= 0.0 THEN Max_RPM_S  := 3000.0; END_IF; (* Trục Dầu S:     Max 3000 RPM *)
IF Max_RPM_T  <= 0.0 THEN Max_RPM_T  := 1500.0; END_IF; (* Trục Thu T:     Max 1500 RPM *)

(* ---------------------------------------------------------------------------- *)
(* 2. KHỞI TẠO TỶ SỐ TRUYỀN HỘP SỐ THỰC TẾ (GEAR RATIO - REAL)                *)
(* ---------------------------------------------------------------------------- *)
IF Gear_Ratio_T  <= 0.0 THEN Gear_Ratio_T  := 10.1; END_IF; (* Thu T:     10.1 : 1 (D620) *)
IF Gear_Ratio_X1 <= 0.0 THEN Gear_Ratio_X1 := 8.0;  END_IF; (* Xả X1:     8.0  : 1 (D622) *)
IF Gear_Ratio_X2 <= 0.0 THEN Gear_Ratio_X2 := 8.0;  END_IF; (* Master X2: 8.0  : 1 (D624) *)
IF Gear_Ratio_Ms <= 0.0 THEN Gear_Ratio_Ms := 10.0; END_IF; (* Ghép Ms:   10.0 : 1 (D626) *)
IF Gear_Ratio_S  <= 0.0 THEN Gear_Ratio_S  := 10.0; END_IF; (* Dầu S:     10.0 : 1 (D628) *)
IF Gear_Ratio_U  <= 0.0 THEN Gear_Ratio_U  := 1.03125; END_IF; (* Trục Xả Metalize U: Gear = 33/32 = 1.03125 (D210) *)

(* ---------------------------------------------------------------------------- *)
(* 3. KHỞI TẠO ĐƯỜNG KÍNH LÔ CƠ CẤU (ROLLER DIAMETER - mm - REAL)              *)
(* ---------------------------------------------------------------------------- *)
IF Dia_X1_Roller_mm <= 0.0 THEN Dia_X1_Roller_mm := 300.5; END_IF; (* Lô Kéo X1:    300.5 mm (D638) *)
IF Dia_X2_Roller_mm <= 0.0 THEN Dia_X2_Roller_mm := 300.5; END_IF; (* Lô Master X2: 300.5 mm (D642) *)
IF Dia_Ms_Roller_mm <= 0.0 THEN Dia_Ms_Roller_mm := 200.0; END_IF; (* Lô Ghép Ms:   200.0 mm (D640) *)
IF Dia_S_Roller_mm  <= 0.0 THEN Dia_S_Roller_mm  := 100.0; END_IF; (* Lô Dầu S:     100.0 mm (D648) *)

(* ---------------------------------------------------------------------------- *)
(* 4. KHỞI TẠO ĐƯỜNG KÍNH LÕI (CORE) VÀ ĐƯỜNG KÍNH MAX (MAX DIA) (mm - REAL)    *)
(* ---------------------------------------------------------------------------- *)
IF Core_Dia_T_mm <= 0.0 THEN Core_Dia_T_mm := 76.0;   END_IF; (* Lõi cuộn Thu T:  76.0 mm (D644) *)
IF Core_Dia_M_mm <= 0.0 THEN Core_Dia_M_mm := 76.0;   END_IF; (* Lõi cuộn Xả M:   76.0 mm (D645) *)
IF Core_Dia_U_mm <= 0.0 THEN Core_Dia_U_mm := 76.0;   END_IF; (* Lõi cuộn Xả U:   76.0 mm (D647) *)

IF Max_Dia_T_mm  <= 0.0 THEN Max_Dia_T_mm  := 1000.0; END_IF; (* Cuộn Thu T max: 1000.0 mm (D646) *)
IF Max_Dia_M_mm  <= 0.0 THEN Max_Dia_M_mm  := 600.0;  END_IF; (* Cuộn Xả M max:   600.0 mm (D649) *)
IF Max_Dia_U_mm  <= 0.0 THEN Max_Dia_U_mm  := 800.0;  END_IF; (* Cuộn Xả U max:   800.0 mm (D650) *)

(* ---------------------------------------------------------------------------- *)
(* 5. KHỞI TẠO ĐƯỜNG KÍNH BAN ĐẦU KHI MỚI BẬT NGUỒN (REAL)                     *)
(* ---------------------------------------------------------------------------- *)
IF Real_Dia_T_mm < Core_Dia_T_mm OR Real_Dia_T_mm > Max_Dia_T_mm THEN
    Real_Dia_T_mm := Core_Dia_T_mm; (* 76.0 mm - D724 *)
END_IF;

IF Real_Dia_M_mm < Core_Dia_M_mm OR Real_Dia_M_mm > Max_Dia_M_mm THEN
    Real_Dia_M_mm := Max_Dia_M_mm;  (* 600.0 mm - D722 *)
END_IF;

IF Real_Dia_U_mm < Core_Dia_U_mm OR Real_Dia_U_mm > Max_Dia_U_mm THEN
    Real_Dia_U_mm := Max_Dia_U_mm;  (* 800.0 mm - D720 *)
END_IF;

(* ---------------------------------------------------------------------------- *)
(* 6. KHỞI TẠO TỶ LỆ TỐC ĐỘ VÀ BÙ TỐC (SPEED RATIO - REAL, 1.0 = 100%)         *)
(* ---------------------------------------------------------------------------- *)
IF Speed_Ratio_T  <= 0.0 THEN Speed_Ratio_T  := 1.05; END_IF; (* Chạy nhanh hơn 5% giữ căng (D756) *)
IF Speed_Ratio_X1 <= 0.0 THEN Speed_Ratio_X1 := 1.00; END_IF; (* Đồng bộ 100.0% (D758) *)
IF Speed_Ratio_Ms <= 0.0 THEN Speed_Ratio_Ms := 1.00; END_IF; (* Đồng bộ 100.0% (D762) *)
IF Speed_Ratio_S  <= 0.0 THEN Speed_Ratio_S  := 1.00; END_IF; (* Đồng bộ 100.0% (D766) *)

(* ---------------------------------------------------------------------------- *)
(* 7. KHỞI TẠO GIỚI HẠN TỐC ĐỘ DÂY CHUYỀN (m/phút - REAL)                      *)
(* ---------------------------------------------------------------------------- *)
IF Max_Speed_MPM         <= 0.0 THEN Max_Speed_MPM         := 100.0; END_IF; (* Max 100.0 m/p (D602) *)
IF Min_Speed_MPM         <= 0.0 THEN Min_Speed_MPM         := 2.0;   END_IF; (* Min 2.0 m/p (D603) *)
IF Release_Pen_Speed_MPM <= 0.0 THEN Release_Pen_Speed_MPM := 2.0;   END_IF; (* Tốc độ nhả pen (D604) *)
IF Ramp_Accel_Rate       <= 0.0 THEN Ramp_Accel_Rate       := 0.5;   END_IF; (* Gia tốc tăng tốc (D606) *)
IF Ramp_Decel_Rate       <= 0.0 THEN Ramp_Decel_Rate       := 1.0;   END_IF; (* Gia tốc giảm tốc (D608) *)
IF Decel_Distance_Meters <= 0.0 THEN Decel_Distance_Meters := 50.0;  END_IF; (* Khoảng cách hãm dừng (m) *)

(* ---------------------------------------------------------------------------- *)
(* 8. KHỞI TẠO CÀI ĐẶT LỰC CĂNG (TENSION SP - kg/N - REAL) & HỆ SỐ PID         *)
(* ---------------------------------------------------------------------------- *)
IF SP_Tension_T  <= 0.0 THEN SP_Tension_T  := 15.0; END_IF; (* SP Lực căng Thu T: 15.0 kg (D660) *)
IF SP_Tension_X1 <= 0.0 THEN SP_Tension_X1 := 12.0; END_IF; (* SP Lực căng Xả X1: 12.0 kg (D662) *)
IF SP_Tension_M  <= 0.0 THEN SP_Tension_M  := 10.0; END_IF; (* SP Lực căng Xả M:  10.0 kg (D664) *)
IF SP_Tension_U  <= 0.0 THEN SP_Tension_U  := 10.0; END_IF; (* SP Lực căng Xả U:  10.0 kg (D668) *)

(* Hệ số PID cuộn Thu T *)
IF Kp_T <= 0.0 THEN Kp_T := 1.5; END_IF;
IF Ki_T <= 0.0 THEN Ki_T := 0.2; END_IF;
IF Kd_T <= 0.0 THEN Kd_T := 0.1; END_IF;

(* Hệ số PID cuộn Xả X1 *)
IF Kp_X1 <= 0.0 THEN Kp_X1 := 1.2; END_IF;
IF Ki_X1 <= 0.0 THEN Ki_X1 := 0.15; END_IF;
IF Kd_X1 <= 0.0 THEN Kd_X1 := 0.08; END_IF;

(* Hệ số PID trục Master X2 *)
IF Kp_X2 <= 0.0 THEN Kp_X2 := 1.0; END_IF;
IF Ki_X2 <= 0.0 THEN Ki_X2 := 0.1; END_IF;
IF Kd_X2 <= 0.0 THEN Kd_X2 := 0.05; END_IF;

(* Hệ số PID trục Ghép Ms *)
IF Kp_Ms <= 0.0 THEN Kp_Ms := 1.0; END_IF;
IF Ki_Ms <= 0.0 THEN Ki_Ms := 0.1; END_IF;
IF Kd_Ms <= 0.0 THEN Kd_Ms := 0.05; END_IF;

(* Hệ số PID trục Dầu S *)
IF Kp_S <= 0.0 THEN Kp_S := 1.0; END_IF;
IF Ki_S <= 0.0 THEN Ki_S := 0.1; END_IF;
IF Kd_S <= 0.0 THEN Kd_S := 0.05; END_IF;

(* Hệ số PID cuộn Thắng M *)
IF Kp_M <= 0.0 THEN Kp_M := 1.0; END_IF;
IF Ki_M <= 0.0 THEN Ki_M := 0.1; END_IF;
IF Kd_M <= 0.0 THEN Kd_M := 0.05; END_IF;

(* Hệ số PID cuộn Xả U *)
IF Kp_U <= 0.0 THEN Kp_U := 1.0; END_IF;
IF Ki_U <= 0.0 THEN Ki_U := 0.1; END_IF;
IF Kd_U <= 0.0 THEN Kd_U := 0.05; END_IF;

(* ---------------------------------------------------------------------------- *)
(* 9. KHỞI TẠO TORQUE HÃM MIN / MAX VÀ GIỮ DỪNG MÁY (% - REAL)                 *)
(* ---------------------------------------------------------------------------- *)
IF Min_Torque_M          <= 0.0 THEN Min_Torque_M          := 4.0;  END_IF; (* 4.0 % *)
IF Max_Torque_M          <= 0.0 THEN Max_Torque_M          := 20.0; END_IF; (* 20.0 % *)
IF Init_Holding_Torque_M <= 0.0 THEN Init_Holding_Torque_M := 8.0;  END_IF; (* 8.0 % *)

IF Min_Torque_U          <= 0.0 THEN Min_Torque_U          := 5.0;  END_IF; (* 5.0 % *)
IF Max_Torque_U          <= 0.0 THEN Max_Torque_U          := 25.0; END_IF; (* 25.0 % *)
IF Init_Holding_Torque_U <= 0.0 THEN Init_Holding_Torque_U := 10.0; END_IF; (* 10.0 % *)

(* ---------------------------------------------------------------------------- *)
(* 10. KHỞI TẠO HỆ SỐ GAIN CALIB LOADCELL (REAL)                                *)
(* ---------------------------------------------------------------------------- *)
IF Calib_Gain_T  <= 0.0 THEN Calib_Gain_T  := 1.0; END_IF;
IF Calib_Gain_X1 <= 0.0 THEN Calib_Gain_X1 := 1.0; END_IF;
IF Calib_Gain_M  <= 0.0 THEN Calib_Gain_M  := 1.0; END_IF;
IF Calib_Gain_U  <= 0.0 THEN Calib_Gain_U  := 1.0; END_IF;

(* ---------------------------------------------------------------------------- *)
(* 11. KHỞI TẠO CẤU HÌNH MODULE Q68ADV (SLOT 0 - HEAD ADDRESS H00)             *)
(* ---------------------------------------------------------------------------- *)
(* BFM #0: Cho phép chuyển đổi A/D cả 8 kênh (0 = Enable, 1 = Disable)          *)
U0\G0 := 16#0000; (* Enable toàn bộ CH1..CH8 *)

(* BFM #9 & #10: Cài đặt chế độ lọc trung bình trượt (Moving Average = 16#3333) *)
U0\G9  := 16#3333; (* CH1..CH4: Moving Average *)
U0\G10 := 16#3333; (* CH5..CH8: Moving Average *)

(* BFM #11..#18: Số lượng mẫu trung bình trượt (16 mẫu liên tục)                *)
U0\G11 := 16; (* CH1: Loadcell Thu T *)
U0\G12 := 16; (* CH2: Loadcell Kéo X1 *)
U0\G13 := 16; (* CH3: Loadcell Thắng M *)
U0\G14 := 16; (* CH4: Loadcell Xả U *)
U0\G15 := 16; (* CH5: Analog Tốc độ Servo Trục S *)
U0\G16 := 16; (* CH6: Dự phòng *)
U0\G17 := 16; (* CH7: Dự phòng *)
U0\G18 := 16; (* CH8: Dự phòng *)

(* ---------------------------------------------------------------------------- *)
(* 12. KHỞI TẠO CẤU HÌNH MODULE Q68DAV (SLOT 1 - HEAD ADDRESS H10)             *)
(* ---------------------------------------------------------------------------- *)
(* BFM #0: Cho phép chuyển đổi D/A cả 8 kênh (0 = Enable, 1 = Disable)          *)
U1\G0 := 16#0000; (* Enable D/A cho CH1..CH8 *)

(* BFM #9: Cho phép ngõ ra Analog Output (Bit 0..7: 1 = Output Enable)          *)
U1\G9 := 16#00FF; (* Cho phép xuất áp ra cả 8 kênh *)

(* Bật cờ Y11 hoặc Y10 cho phép chuyển đổi D/A *)
Y11 := TRUE;
END_PROGRAM

// device comments not shown above
D524  ; DAC CH1: Speed Thu T
D526  ; DAC CH3: Speed Xa X1
X50  ; "X","50","Sensor tiem can dem vo
X51  ; "X","51","Sensor tiem can dem vo
SM409  ; 0.01 second clock
M1104  ; Remote Input X0 (St4)
M1105  ; Remote Input X1 (St4)
M1106  ; Remote Input X2 (St4)
M1107  ; Remote Input X3 (St4)
M1108  ; Remote Input X4 (St4)
M1109  ; Remote Input X5 (St4)
M1110  ; Remote Input X6 (St4)
M1111  ; Remote Input X7 (St4)
M1208  ; Cho phép chuyển đổi A/D Trạm 1 (
M1240  ; Cho phép chuyển đổi D/A Trạm 2 (
M1304  ; Servo ON Truc Thu T (Y8)
M1305  ; Servo ON Truc Xa X1 (Y9)
M1306  ; Servo ON Truc Master X2 (YA)
M1307  ; Servo ON Truc Ghep Ms (YB)
M1308  ; Servo ON Truc Trang Dau S (YC)
M1309  ; Solenoid Valve Pen 1 (YD)
M1310  ; Solenoid Valve Pen 2 (YE)
M1311  ; Du phong / Bao loi (YF)
D525  ; DAC CH2: Torque Thu T
D527  ; DAC CH4: Speed Master X2
D528  ; DAC CH5: Speed Ghep Ms
D529  ; DAC CH6: Torque Ghep Ms
D530  ; DAC CH7: Speed Trang Dau S
D531  ; DAC CH8: Speed Xa U
X52  ; "X","52","Nut nhan START vat ly
X53  ; "X","53","Nut nhan STOP vat ly (
X54  ; "X","54","Nut nhan INC Tang toc
X55  ; "X","55","Nut nhan DEC Giam toc
X56  ; "X","56","Nut Toggle Pen 1 vat l
X57  ; "X","57","Nut Toggle Pen 2 vat l
X58  ; "X","58","Cong tac Giu Torque M
X59  ; "X","59","Cong tac Giu Torque U
X5A  ; "X","5A","Cong tac Rua may bo ch
X5B  ; "X","5B","Cong tac Rua may bo ch
X5C  ; "X","5C","Nut nhan co BO CHAM NO
